(* Control logic *)
IF CtrlExton THEN
	REL_EN:=TRUE;
ELSE
	CASE CTRL_MODE OF
		 0: REL_EN:=FALSE;
		-1: REL_EN:=TRUE;
		-2: REL_EN:=CtrlKey;
		-3: REL_EN:=NOT CtrlKey;
		-4: REL_EN:=CtrlSens;
		-5: REL_EN:=NOT CtrlSens;
	ELSE
		IF CTRL_MODE>0 THEN
			REL_EN:=TrigTimer.Q;
			TrigTimer.PT:=T#1S*CTRL_MODE;
		ELSE
			REL_EN:=FALSE;
		END_IF
	END_CASE
END_IF

(* Temporary energy counter *)
TickTimer(IN:=NOT TickTimer.Q);
IF TickTimer.Q AND REL_EN THEN
	WORKINGTIME:=WORKINGTIME+1;
	ENERGYCOUNTER_T:=ENERGYCOUNTER_T+REL_V*REL_A;
	IF ENERGYCOUNTER_T>36000000 THEN
		ENERGYCOUNTER_T:=ENERGYCOUNTER_T-36000000;
		ENERGYCOUNTER:=ENERGYCOUNTER+1;		
	END_IF
END_IF

(* Generate status events *)
sREL_EN(IN:=REL_EN);
IF sREL_EN.EVL THEN LogEv(EL_Log,EO_LUXM,ID,2,''); END_IF
IF sREL_EN.EVH THEN LogEv(EL_Log,EO_LUXM,ID,3,''); POWERONCYCLES:=POWERONCYCLES+1; END_IF

(* Check status feedback *)
chkREL_ST(IN:=(REL_ST<>REL_EN));
IF chkREL_ST.EVH THEN LogEv(EL_Alarm,EO_LUXM,ID,9,''); END_IF
IF chkREL_ST.EVL AND sREL_ALM=0 THEN LogEv(EL_Log,EO_LUXM,ID,1,''); END_IF

(* Check controller alarm *)
IF sREL_ALM<>REL_ALM THEN
	CASE REL_ALM OF
		0: IF NOT chkREL_ST.OUT THEN LogEv(EL_Log,EO_LUXM,ID,1,''); END_IF
		1: LogEv(EL_Alarm,EO_LUXM,ID,6,'');
		2: LogEv(EL_Wrn  ,EO_LUXM,ID,4,WORD_TO_STRING(REL_A));
		3: LogEv(EL_Wrn  ,EO_LUXM,ID,5,WORD_TO_STRING(REL_A));
		4: LogEv(EL_Alarm,EO_LUXM,ID,7,WORD_TO_STRING(REL_A));
		5: LogEv(EL_Alarm,EO_LUXM,ID,8,'');
	END_CASE
	sREL_ALM:=REL_ALM;
END_IF

(* Status color *)
   IF REL_ALM=1 OR REL_ALM>3 OR chkREL_ST.OUT	THEN Status_Log:=2; Status_Vis:=COLOR_RED;
ELSIF REL_ALM<>0								THEN Status_Log:=1; Status_Vis:=COLOR_YELLOW;
                  	   							ELSE Status_Log:=0; Status_Vis:=SEL(REL_EN,COLOR_GREEN_OFF,COLOR_GREEN);
END_IF

ACTION AddLogData:
Logger.s1:=INSERT('&LUXM=',BYTE_TO_STRING(ID),5);
IF ID<10 THEN Logger.s1:=INSERT(Logger.s1,'0',5); END_IF

Logger.s1:=CONCAT(Logger.s1,WORD_TO_STRING(REL_V));				Logger.s1:=CONCAT(Logger.s1,';');
Logger.s1:=CONCAT(Logger.s1,WORD_TO_STRING(REL_A));				Logger.s1:=CONCAT(Logger.s1,';');
Logger.s1:=CONCAT(Logger.s1,DWORD_TO_STRING(ENERGYCOUNTER));	Logger.s1:=CONCAT(Logger.s1,';');
Logger.s1:=CONCAT(Logger.s1,DWORD_TO_STRING(WORKINGTIME));		Logger.s1:=CONCAT(Logger.s1,';');
Logger.s1:=CONCAT(Logger.s1,DWORD_TO_STRING(POWERONCYCLES));	Logger.s1:=CONCAT(Logger.s1,';');
Logger.s1:=CONCAT(Logger.s1,INT_TO_STRING(REL_TEMP));			Logger.s1:=CONCAT(Logger.s1,';');

Logger.s1:=CONCAT(Logger.s1,BYTE_TO_STRING(Status_Log));
ADDSTRING(ADR(Logger.TData), ADR(Logger.s1), Logger.TLen);
END_ACTION

ACTION StatReset:
(* Reset statistic counters *)
WORKINGTIME:=0;
POWERONCYCLES:=0;
ENERGYCOUNTER:=0;
END_ACTION

END_FUNCTION_BLOCK

// Utils Functions/DirOpen_FB
FUNCTION_BLOCK DirOpen_FB
VAR_INPUT
END_VAR
VAR_OUTPUT
END_VAR
VAR
	iFilesCount, counter : word;
//	DirNames: array[1..64] of string;
//	FileNames: array[1..64] of string;
	
	sDirName : STRING;
	sDirEntry : STRING;
	udiDirHandle : RTS_IEC_HANDLE;
	stDirInfo : DirInfo;
	udiResult : __XWORD;
	udiCreateError: UDINT;
	udiReadError: UDINT;
END_VAR

(*
sDirName:='Pippo';
udiCreateError := SysDirCreate(szDir:= sDirName);
*)

//ConfPath:='/media/sd/';	
sDirName:=CONCAT(STR1:=ConfPath, STR2:=sDirName);
udiDirHandle := SysDirOpen(szDir:= sDirName, szDirEntry:= sDirEntry, diMaxDirEntry:= 1024,
				pDirInfo:= ADR(stDirInfo), pResult:= udiResult);

(* Iterate through all direcotry entries and count them. The implicit entries with points are not count.
when the last entry is reached the SysDirRead always delivers the last entry.*)
iFilesCount := 0;
counter := 1;
repeat
	if FIND(sDirEntry, '.') <> 1 then
		iFilesCount := iFilesCount +1;
	end_if
	udiReadError:= SysDirRead(hDir:= udiDirHandle, szDirEntry:= sDirEntry, diMaxDirEntry:= 1024, pDirInfo:=ADR(stDirInfo) );
	// SysDirRead is used to Directory Info
	// Here, Im using SysDirRead to Find Folder Names within a Directory
	// If stDirInfo.diDirectory is Hex 2 , then the Directory is a folder, otherwise Hex 0 is a File
	if stDirInfo.diDirectory = 16#2 and Find(sDirEntry,'.') <> 1 then
		DirNames[counter]:=sDirEntry;
	else
		FileNames[counter]:=sDirEntry;
	counter:=counter+1;
	end_if
until 
	udiReadError = CmpErrors.Errors.ERR_END_OF_OBJECT
end_repeat

END_FUNCTION_BLOCK

// AC14nn/Application/VIS_CHONOEDITOR
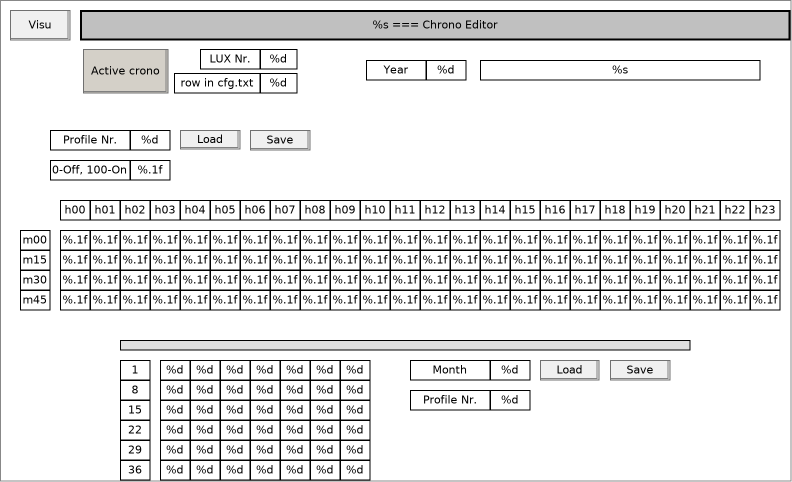
VISUALIZATION VIS_CHONOEDITOR  // 792x482
VAR_IN_OUT
//	x	: word;
//	LuxSel	: word;	
END_VAR
    Rectangle (200,49 60x20), "LUX Nr."
    Rectangle (260,49 37x20), "%d", text variable: CronEd.CN_Sel, colour toggle: CronEd.CN_Sel<>CronEd.CN_Act
        OnMouseDown: write the text variable via Edit, min 1, max 900, title '1'
    Rectangle (50,130 80x20), "Profile Nr."
    Rectangle (130,130 40x20), "%d", text variable: CronEd.PR_Sel, colour toggle: CronEd.PR_Sel<>CronEd.PR_Act
        OnMouseDown: write the text variable via Edit, min 1, max 10
    Rectangle (50,160 80x20), "0-Off, 100-On"
    Rectangle (130,160 40x20), "%.1f", text variable: CronEd.PR_TT
        OnMouseDown: write the text variable via Edit
    Button (180,130 60x19), "Load", pressed state: CronEd.PR_Load
        toggle CronEd.PR_Load
    Button (250,130 60x20), "Save", pressed state: CronEd.PR_Save
        toggle CronEd.PR_Save
    Rectangle (20,230 30x20), "m00"
    Rectangle (20,250 30x20), "m15"
    Rectangle (20,270 30x20), "m30"
    Rectangle (20,290 30x20), "m45"
    Rectangle (80,10 710x30), "%s === Chrono Editor", text variable: Plant_NAME
    Button (10,10 60x30), "Visu"
        OnMouseUp:  Assign=PLC_Visualization, Type=Assignment
    Polygon (20,210)
    RoundedRectangle (60,230 30x20), "%.1f", text variable: INT_TO_REAL(CronEd.PR.Setpoint[0])/10
        OnMouseUp: execute { CronEd.PR.Setpoint[0]:=(REAL_TO_WORD(CronEd.PR_TT*10)); }
    RoundedRectangle (60,250 30x20), "%.1f", text variable: INT_TO_REAL(CronEd.PR.Setpoint[1])/10
        OnMouseUp: execute { CronEd.PR.Setpoint[1]:=(REAL_TO_WORD(CronEd.PR_TT*10)); }
    RoundedRectangle (60,270 30x20), "%.1f", text variable: INT_TO_REAL(CronEd.PR.Setpoint[2])/10
        OnMouseUp: execute { CronEd.PR.Setpoint[2]:=(REAL_TO_WORD(CronEd.PR_TT*10)); }
    RoundedRectangle (60,290 30x20), "%.1f", text variable: INT_TO_REAL(CronEd.PR.Setpoint[3])/10
        OnMouseUp: execute { CronEd.PR.Setpoint[3]:=(REAL_TO_WORD(CronEd.PR_TT*10)); }
    Rectangle (60,200 30x20), "h00"
        OnMouseUp: execute { CronEd.PR.Setpoint[0]:=(REAL_TO_WORD(CronEd.PR_TT*10)); }
        OnMouseUp: execute { CronEd.PR.Setpoint[1]:=(REAL_TO_WORD(CronEd.PR_TT*10)); }
        OnMouseUp: execute { CronEd.PR.Setpoint[2]:=(REAL_TO_WORD(CronEd.PR_TT*10)); }
        OnMouseUp: execute { CronEd.PR.Setpoint[3]:=(REAL_TO_WORD(CronEd.PR_TT*10)); }
    RoundedRectangle (90,230 30x20), "%.1f", text variable: INT_TO_REAL(CronEd.PR.Setpoint[4])/10
        OnMouseUp: execute { CronEd.PR.Setpoint[4]:=(REAL_TO_WORD(CronEd.PR_TT*10)); }
    RoundedRectangle (90,250 30x20), "%.1f", text variable: INT_TO_REAL(CronEd.PR.Setpoint[5])/10
        OnMouseUp: execute { CronEd.PR.Setpoint[5]:=(REAL_TO_WORD(CronEd.PR_TT*10)); }
    RoundedRectangle (90,270 30x20), "%.1f", text variable: INT_TO_REAL(CronEd.PR.Setpoint[6])/10
        OnMouseUp: execute { CronEd.PR.Setpoint[6]:=(REAL_TO_WORD(CronEd.PR_TT*10)); }
    RoundedRectangle (90,290 30x20), "%.1f", text variable: INT_TO_REAL(CronEd.PR.Setpoint[7])/10
        OnMouseUp: execute { CronEd.PR.Setpoint[7]:=(REAL_TO_WORD(CronEd.PR_TT*10)); }
    Rectangle (90,200 30x20), "h01"
        OnMouseUp: execute { CronEd.PR.Setpoint[4]:=(REAL_TO_WORD(CronEd.PR_TT*10)); }
        OnMouseUp: execute { CronEd.PR.Setpoint[5]:=(REAL_TO_WORD(CronEd.PR_TT*10)); }
        OnMouseUp: execute { CronEd.PR.Setpoint[6]:=(REAL_TO_WORD(CronEd.PR_TT*10)); }
        OnMouseUp: execute { CronEd.PR.Setpoint[7]:=(REAL_TO_WORD(CronEd.PR_TT*10)); }
    RoundedRectangle (120,230 30x20), "%.1f", text variable: INT_TO_REAL(CronEd.PR.Setpoint[8])/10
        OnMouseUp: execute { CronEd.PR.Setpoint[8]:=(REAL_TO_WORD(CronEd.PR_TT*10)); }
    RoundedRectangle (120,250 30x20), "%.1f", text variable: INT_TO_REAL(CronEd.PR.Setpoint[9])/10
        OnMouseUp: execute { CronEd.PR.Setpoint[9]:=(REAL_TO_WORD(CronEd.PR_TT*10)); }
    RoundedRectangle (120,270 30x20), "%.1f", text variable: INT_TO_REAL(CronEd.PR.Setpoint[10])/10
        OnMouseUp: execute { CronEd.PR.Setpoint[10]:=(REAL_TO_WORD(CronEd.PR_TT*10)); }
    RoundedRectangle (120,290 30x20), "%.1f", text variable: INT_TO_REAL(CronEd.PR.Setpoint[11])/10
        OnMouseUp: execute { CronEd.PR.Setpoint[11]:=(REAL_TO_WORD(CronEd.PR_TT*10)); }
    Rectangle (120,200 30x20), "h02"
        OnMouseUp: execute { CronEd.PR.Setpoint[8]:=(REAL_TO_WORD(CronEd.PR_TT*10)); }
        OnMouseUp: execute { CronEd.PR.Setpoint[9]:=(REAL_TO_WORD(CronEd.PR_TT*10)); }
        OnMouseUp: execute { CronEd.PR.Setpoint[10]:=(REAL_TO_WORD(CronEd.PR_TT*10)); }
        OnMouseUp: execute { CronEd.PR.Setpoint[11]:=(REAL_TO_WORD(CronEd.PR_TT*10)); }
    RoundedRectangle (150,230 30x20), "%.1f", text variable: INT_TO_REAL(CronEd.PR.Setpoint[12])/10
        OnMouseUp: execute { CronEd.PR.Setpoint[12]:=(REAL_TO_WORD(CronEd.PR_TT*10)); }
    RoundedRectangle (150,250 30x20), "%.1f", text variable: INT_TO_REAL(CronEd.PR.Setpoint[13])/10
        OnMouseUp: execute { CronEd.PR.Setpoint[13]:=(REAL_TO_WORD(CronEd.PR_TT*10)); }
    RoundedRectangle (150,270 30x20), "%.1f", text variable: INT_TO_REAL(CronEd.PR.Setpoint[14])/10
        OnMouseUp: execute { CronEd.PR.Setpoint[14]:=(REAL_TO_WORD(CronEd.PR_TT*10)); }
    RoundedRectangle (150,290 30x20), "%.1f", text variable: INT_TO_REAL(CronEd.PR.Setpoint[15])/10
        OnMouseUp: execute { CronEd.PR.Setpoint[15]:=(REAL_TO_WORD(CronEd.PR_TT*10)); }
    Rectangle (150,200 30x20), "h03"
        OnMouseUp: execute { CronEd.PR.Setpoint[15]:=(REAL_TO_WORD(CronEd.PR_TT*10)); }
        OnMouseUp: execute { CronEd.PR.Setpoint[14]:=(REAL_TO_WORD(CronEd.PR_TT*10)); }
        OnMouseUp: execute { CronEd.PR.Setpoint[13]:=(REAL_TO_WORD(CronEd.PR_TT*10)); }
        OnMouseUp: execute { CronEd.PR.Setpoint[12]:=(REAL_TO_WORD(CronEd.PR_TT*10)); }
    RoundedRectangle (180,230 30x20), "%.1f", text variable: INT_TO_REAL(CronEd.PR.Setpoint[16])/10
        OnMouseUp: execute { CronEd.PR.Setpoint[16]:=(REAL_TO_WORD(CronEd.PR_TT*10)); }
    RoundedRectangle (180,250 30x20), "%.1f", text variable: INT_TO_REAL(CronEd.PR.Setpoint[17])/10
        OnMouseUp: execute { CronEd.PR.Setpoint[17]:=(REAL_TO_WORD(CronEd.PR_TT*10)); }
    RoundedRectangle (180,270 30x20), "%.1f", text variable: INT_TO_REAL(CronEd.PR.Setpoint[18])/10
        OnMouseUp: execute { CronEd.PR.Setpoint[18]:=(REAL_TO_WORD(CronEd.PR_TT*10)); }
    RoundedRectangle (180,290 30x20), "%.1f", text variable: INT_TO_REAL(CronEd.PR.Setpoint[19])/10
        OnMouseUp: execute { CronEd.PR.Setpoint[19]:=(REAL_TO_WORD(CronEd.PR_TT*10)); }
    Rectangle (180,200 30x20), "h04"
        OnMouseUp: execute { CronEd.PR.Setpoint[19]:=(REAL_TO_WORD(CronEd.PR_TT*10)); }
        OnMouseUp: execute { CronEd.PR.Setpoint[18]:=(REAL_TO_WORD(CronEd.PR_TT*10)); }
        OnMouseUp: execute { CronEd.PR.Setpoint[17]:=(REAL_TO_WORD(CronEd.PR_TT*10)); }
        OnMouseUp: execute { CronEd.PR.Setpoint[16]:=(REAL_TO_WORD(CronEd.PR_TT*10)); }
    RoundedRectangle (210,230 30x20), "%.1f", text variable: INT_TO_REAL(CronEd.PR.Setpoint[20])/10
        OnMouseUp: execute { CronEd.PR.Setpoint[20]:=(REAL_TO_WORD(CronEd.PR_TT*10)); }
    RoundedRectangle (210,250 30x20), "%.1f", text variable: INT_TO_REAL(CronEd.PR.Setpoint[21])/10
        OnMouseUp: execute { CronEd.PR.Setpoint[21]:=(REAL_TO_WORD(CronEd.PR_TT*10)); }
    RoundedRectangle (210,270 30x20), "%.1f", text variable: INT_TO_REAL(CronEd.PR.Setpoint[22])/10
        OnMouseUp: execute { CronEd.PR.Setpoint[22]:=(REAL_TO_WORD(CronEd.PR_TT*10)); }
    RoundedRectangle (210,290 30x20), "%.1f", text variable: INT_TO_REAL(CronEd.PR.Setpoint[23])/10
        OnMouseUp: execute { CronEd.PR.Setpoint[23]:=(REAL_TO_WORD(CronEd.PR_TT*10)); }
    Rectangle (210,200 30x20), "h05"
        OnMouseUp: execute { CronEd.PR.Setpoint[23]:=(REAL_TO_WORD(CronEd.PR_TT*10)); }
        OnMouseUp: execute { CronEd.PR.Setpoint[22]:=(REAL_TO_WORD(CronEd.PR_TT*10)); }
        OnMouseUp: execute { CronEd.PR.Setpoint[21]:=(REAL_TO_WORD(CronEd.PR_TT*10)); }
        OnMouseUp: execute { CronEd.PR.Setpoint[20]:=(REAL_TO_WORD(CronEd.PR_TT*10)); }
    RoundedRectangle (240,230 30x20), "%.1f", text variable: INT_TO_REAL(CronEd.PR.Setpoint[24])/10
        OnMouseUp: execute { CronEd.PR.Setpoint[24]:=(REAL_TO_WORD(CronEd.PR_TT*10)); }
    RoundedRectangle (240,250 30x20), "%.1f", text variable: INT_TO_REAL(CronEd.PR.Setpoint[25])/10
        OnMouseUp: execute { CronEd.PR.Setpoint[25]:=(REAL_TO_WORD(CronEd.PR_TT*10)); }
    RoundedRectangle (240,270 30x20), "%.1f", text variable: INT_TO_REAL(CronEd.PR.Setpoint[26])/10
        OnMouseUp: execute { CronEd.PR.Setpoint[26]:=(REAL_TO_WORD(CronEd.PR_TT*10)); }
    RoundedRectangle (240,290 30x20), "%.1f", text variable: INT_TO_REAL(CronEd.PR.Setpoint[27])/10
        OnMouseUp: execute { CronEd.PR.Setpoint[27]:=(REAL_TO_WORD(CronEd.PR_TT*10)); }
    Rectangle (240,200 30x20), "h06"
        OnMouseUp: execute { CronEd.PR.Setpoint[27]:=(REAL_TO_WORD(CronEd.PR_TT*10)); }
        OnMouseUp: execute { CronEd.PR.Setpoint[26]:=(REAL_TO_WORD(CronEd.PR_TT*10)); }
        OnMouseUp: execute { CronEd.PR.Setpoint[25]:=(REAL_TO_WORD(CronEd.PR_TT*10)); }
        OnMouseUp: execute { CronEd.PR.Setpoint[24]:=(REAL_TO_WORD(CronEd.PR_TT*10)); }
    RoundedRectangle (270,230 30x20), "%.1f", text variable: INT_TO_REAL(CronEd.PR.Setpoint[28])/10
        OnMouseUp: execute { CronEd.PR.Setpoint[28]:=(REAL_TO_WORD(CronEd.PR_TT*10)); }
    RoundedRectangle (270,250 30x20), "%.1f", text variable: INT_TO_REAL(CronEd.PR.Setpoint[29])/10
        OnMouseUp: execute { CronEd.PR.Setpoint[29]:=(REAL_TO_WORD(CronEd.PR_TT*10)); }
    RoundedRectangle (270,270 30x20), "%.1f", text variable: INT_TO_REAL(CronEd.PR.Setpoint[30])/10
        OnMouseUp: execute { CronEd.PR.Setpoint[30]:=(REAL_TO_WORD(CronEd.PR_TT*10)); }
    RoundedRectangle (270,290 30x20), "%.1f", text variable: INT_TO_REAL(CronEd.PR.Setpoint[31])/10
        OnMouseUp: execute { CronEd.PR.Setpoint[31]:=(REAL_TO_WORD(CronEd.PR_TT*10)); }
    Rectangle (270,200 30x20), "h07"
        OnMouseUp: execute { CronEd.PR.Setpoint[31]:=(REAL_TO_WORD(CronEd.PR_TT*10)); }
        OnMouseUp: execute { CronEd.PR.Setpoint[30]:=(REAL_TO_WORD(CronEd.PR_TT*10)); }
        OnMouseUp: execute { CronEd.PR.Setpoint[29]:=(REAL_TO_WORD(CronEd.PR_TT*10)); }
        OnMouseUp: execute { CronEd.PR.Setpoint[28]:=(REAL_TO_WORD(CronEd.PR_TT*10)); }
    RoundedRectangle (300,230 30x20), "%.1f", text variable: INT_TO_REAL(CronEd.PR.Setpoint[32])/10
        OnMouseUp: execute { CronEd.PR.Setpoint[32]:=(REAL_TO_WORD(CronEd.PR_TT*10)); }
    RoundedRectangle (300,250 30x20), "%.1f", text variable: INT_TO_REAL(CronEd.PR.Setpoint[33])/10
        OnMouseUp: execute { CronEd.PR.Setpoint[33]:=(REAL_TO_WORD(CronEd.PR_TT*10)); }
    RoundedRectangle (300,270 30x20), "%.1f", text variable: INT_TO_REAL(CronEd.PR.Setpoint[34])/10
        OnMouseUp: execute { CronEd.PR.Setpoint[34]:=(REAL_TO_WORD(CronEd.PR_TT*10)); }
    RoundedRectangle (300,290 30x20), "%.1f", text variable: INT_TO_REAL(CronEd.PR.Setpoint[35])/10
        OnMouseUp: execute { CronEd.PR.Setpoint[35]:=(REAL_TO_WORD(CronEd.PR_TT*10)); }
    Rectangle (300,200 30x20), "h08"
        OnMouseUp: execute { CronEd.PR.Setpoint[35]:=(REAL_TO_WORD(CronEd.PR_TT*10)); }
        OnMouseUp: execute { CronEd.PR.Setpoint[34]:=(REAL_TO_WORD(CronEd.PR_TT*10)); }
        OnMouseUp: execute { CronEd.PR.Setpoint[33]:=(REAL_TO_WORD(CronEd.PR_TT*10)); }
        OnMouseUp: execute { CronEd.PR.Setpoint[32]:=(REAL_TO_WORD(CronEd.PR_TT*10)); }
    RoundedRectangle (330,230 30x20), "%.1f", text variable: INT_TO_REAL(CronEd.PR.Setpoint[36])/10
        OnMouseUp: execute { CronEd.PR.Setpoint[36]:=(REAL_TO_WORD(CronEd.PR_TT*10)); }
    RoundedRectangle (330,250 30x20), "%.1f", text variable: INT_TO_REAL(CronEd.PR.Setpoint[37])/10
        OnMouseUp: execute { CronEd.PR.Setpoint[37]:=(REAL_TO_WORD(CronEd.PR_TT*10)); }
    RoundedRectangle (330,270 30x20), "%.1f", text variable: INT_TO_REAL(CronEd.PR.Setpoint[38])/10
        OnMouseUp: execute { CronEd.PR.Setpoint[38]:=(REAL_TO_WORD(CronEd.PR_TT*10)); }
    RoundedRectangle (330,290 30x20), "%.1f", text variable: INT_TO_REAL(CronEd.PR.Setpoint[39])/10
        OnMouseUp: execute { CronEd.PR.Setpoint[39]:=(REAL_TO_WORD(CronEd.PR_TT*10)); }
    Rectangle (330,200 30x20), "h09"
        OnMouseUp: execute { CronEd.PR.Setpoint[39]:=(REAL_TO_WORD(CronEd.PR_TT*10)); }
        OnMouseUp: execute { CronEd.PR.Setpoint[38]:=(REAL_TO_WORD(CronEd.PR_TT*10)); }
        OnMouseUp: execute { CronEd.PR.Setpoint[37]:=(REAL_TO_WORD(CronEd.PR_TT*10)); }
        OnMouseUp: execute { CronEd.PR.Setpoint[36]:=(REAL_TO_WORD(CronEd.PR_TT*10)); }
    RoundedRectangle (360,230 30x20), "%.1f", text variable: INT_TO_REAL(CronEd.PR.Setpoint[40])/10
        OnMouseUp: execute { CronEd.PR.Setpoint[40]:=(REAL_TO_WORD(CronEd.PR_TT*10)); }
    RoundedRectangle (360,250 30x20), "%.1f", text variable: INT_TO_REAL(CronEd.PR.Setpoint[41])/10
        OnMouseUp: execute { CronEd.PR.Setpoint[41]:=(REAL_TO_WORD(CronEd.PR_TT*10)); }
    RoundedRectangle (360,270 30x20), "%.1f", text variable: INT_TO_REAL(CronEd.PR.Setpoint[42])/10
        OnMouseUp: execute { CronEd.PR.Setpoint[42]:=(REAL_TO_WORD(CronEd.PR_TT*10)); }
    RoundedRectangle (360,290 30x20), "%.1f", text variable: INT_TO_REAL(CronEd.PR.Setpoint[43])/10
        OnMouseUp: execute { CronEd.PR.Setpoint[43]:=(REAL_TO_WORD(CronEd.PR_TT*10)); }
    Rectangle (360,200 30x20), "h10"
        OnMouseUp: execute { CronEd.PR.Setpoint[43]:=(REAL_TO_WORD(CronEd.PR_TT*10)); }
        OnMouseUp: execute { CronEd.PR.Setpoint[42]:=(REAL_TO_WORD(CronEd.PR_TT*10)); }
        OnMouseUp: execute { CronEd.PR.Setpoint[41]:=(REAL_TO_WORD(CronEd.PR_TT*10)); }
        OnMouseUp: execute { CronEd.PR.Setpoint[40]:=(REAL_TO_WORD(CronEd.PR_TT*10)); }
    RoundedRectangle (390,230 30x20), "%.1f", text variable: INT_TO_REAL(CronEd.PR.Setpoint[44])/10
        OnMouseUp: execute { CronEd.PR.Setpoint[44]:=(REAL_TO_WORD(CronEd.PR_TT*10)); }
    RoundedRectangle (390,250 30x20), "%.1f", text variable: INT_TO_REAL(CronEd.PR.Setpoint[45])/10
        OnMouseUp: execute { CronEd.PR.Setpoint[45]:=(REAL_TO_WORD(CronEd.PR_TT*10)); }
    RoundedRectangle (390,270 30x20), "%.1f", text variable: INT_TO_REAL(CronEd.PR.Setpoint[46])/10
        OnMouseUp: execute { CronEd.PR.Setpoint[46]:=(REAL_TO_WORD(CronEd.PR_TT*10)); }
    RoundedRectangle (390,290 30x20), "%.1f", text variable: INT_TO_REAL(CronEd.PR.Setpoint[47])/10
        OnMouseUp: execute { CronEd.PR.Setpoint[47]:=(REAL_TO_WORD(CronEd.PR_TT*10)); }
    Rectangle (390,200 30x20), "h11"
        OnMouseUp: execute { CronEd.PR.Setpoint[47]:=(REAL_TO_WORD(CronEd.PR_TT*10)); }
        OnMouseUp: execute { CronEd.PR.Setpoint[46]:=(REAL_TO_WORD(CronEd.PR_TT*10)); }
        OnMouseUp: execute { CronEd.PR.Setpoint[45]:=(REAL_TO_WORD(CronEd.PR_TT*10)); }
        OnMouseUp: execute { CronEd.PR.Setpoint[44]:=(REAL_TO_WORD(CronEd.PR_TT*10)); }
    RoundedRectangle (420,230 30x20), "%.1f", text variable: INT_TO_REAL(CronEd.PR.Setpoint[48])/10
        OnMouseUp: execute { CronEd.PR.Setpoint[48]:=(REAL_TO_WORD(CronEd.PR_TT*10)); }
    RoundedRectangle (420,250 30x20), "%.1f", text variable: INT_TO_REAL(CronEd.PR.Setpoint[49])/10
        OnMouseUp: execute { CronEd.PR.Setpoint[49]:=(REAL_TO_WORD(CronEd.PR_TT*10)); }
    RoundedRectangle (420,270 30x20), "%.1f", text variable: INT_TO_REAL(CronEd.PR.Setpoint[50])/10
        OnMouseUp: execute { CronEd.PR.Setpoint[50]:=(REAL_TO_WORD(CronEd.PR_TT*10)); }
    RoundedRectangle (420,290 30x20), "%.1f", text variable: INT_TO_REAL(CronEd.PR.Setpoint[51])/10
        OnMouseUp: execute { CronEd.PR.Setpoint[51]:=(REAL_TO_WORD(CronEd.PR_TT*10)); }
    Rectangle (420,200 30x20), "h12"
        OnMouseUp: execute { CronEd.PR.Setpoint[51]:=(REAL_TO_WORD(CronEd.PR_TT*10)); }
        OnMouseUp: execute { CronEd.PR.Setpoint[50]:=(REAL_TO_WORD(CronEd.PR_TT*10)); }
        OnMouseUp: execute { CronEd.PR.Setpoint[49]:=(REAL_TO_WORD(CronEd.PR_TT*10)); }
        OnMouseUp: execute { CronEd.PR.Setpoint[48]:=(REAL_TO_WORD(CronEd.PR_TT*10)); }
    RoundedRectangle (450,230 30x20), "%.1f", text variable: INT_TO_REAL(CronEd.PR.Setpoint[52])/10
        OnMouseUp: execute { CronEd.PR.Setpoint[52]:=(REAL_TO_WORD(CronEd.PR_TT*10)); }
    RoundedRectangle (450,250 30x20), "%.1f", text variable: INT_TO_REAL(CronEd.PR.Setpoint[53])/10
        OnMouseUp: execute { CronEd.PR.Setpoint[53]:=(REAL_TO_WORD(CronEd.PR_TT*10)); }
    RoundedRectangle (450,270 30x20), "%.1f", text variable: INT_TO_REAL(CronEd.PR.Setpoint[54])/10
        OnMouseUp: execute { CronEd.PR.Setpoint[54]:=(REAL_TO_WORD(CronEd.PR_TT*10)); }
    RoundedRectangle (450,290 30x20), "%.1f", text variable: INT_TO_REAL(CronEd.PR.Setpoint[55])/10
        OnMouseUp: execute { CronEd.PR.Setpoint[55]:=(REAL_TO_WORD(CronEd.PR_TT*10)); }
    Rectangle (450,200 30x20), "h13"
        OnMouseUp: execute { CronEd.PR.Setpoint[55]:=(REAL_TO_WORD(CronEd.PR_TT*10)); }
        OnMouseUp: execute { CronEd.PR.Setpoint[54]:=(REAL_TO_WORD(CronEd.PR_TT*10)); }
        OnMouseUp: execute { CronEd.PR.Setpoint[53]:=(REAL_TO_WORD(CronEd.PR_TT*10)); }
        OnMouseUp: execute { CronEd.PR.Setpoint[52]:=(REAL_TO_WORD(CronEd.PR_TT*10)); }
    RoundedRectangle (480,230 30x20), "%.1f", text variable: INT_TO_REAL(CronEd.PR.Setpoint[56])/10
        OnMouseUp: execute { CronEd.PR.Setpoint[56]:=(REAL_TO_WORD(CronEd.PR_TT*10)); }
    RoundedRectangle (480,250 30x20), "%.1f", text variable: INT_TO_REAL(CronEd.PR.Setpoint[57])/10
        OnMouseUp: execute { CronEd.PR.Setpoint[57]:=(REAL_TO_WORD(CronEd.PR_TT*10)); }
    RoundedRectangle (480,270 30x20), "%.1f", text variable: INT_TO_REAL(CronEd.PR.Setpoint[58])/10
        OnMouseUp: execute { CronEd.PR.Setpoint[58]:=(REAL_TO_WORD(CronEd.PR_TT*10)); }
    RoundedRectangle (480,290 30x20), "%.1f", text variable: INT_TO_REAL(CronEd.PR.Setpoint[59])/10
        OnMouseUp: execute { CronEd.PR.Setpoint[59]:=(REAL_TO_WORD(CronEd.PR_TT*10)); }
    Rectangle (480,200 30x20), "h14"
        OnMouseUp: execute { CronEd.PR.Setpoint[59]:=(REAL_TO_WORD(CronEd.PR_TT*10)); }
        OnMouseUp: execute { CronEd.PR.Setpoint[58]:=(REAL_TO_WORD(CronEd.PR_TT*10)); }
        OnMouseUp: execute { CronEd.PR.Setpoint[57]:=(REAL_TO_WORD(CronEd.PR_TT*10)); }
        OnMouseUp: execute { CronEd.PR.Setpoint[56]:=(REAL_TO_WORD(CronEd.PR_TT*10)); }
    RoundedRectangle (510,230 30x20), "%.1f", text variable: INT_TO_REAL(CronEd.PR.Setpoint[60])/10
        OnMouseUp: execute { CronEd.PR.Setpoint[60]:=(REAL_TO_WORD(CronEd.PR_TT*10)); }
    RoundedRectangle (510,250 30x20), "%.1f", text variable: INT_TO_REAL(CronEd.PR.Setpoint[61])/10
        OnMouseUp: execute { CronEd.PR.Setpoint[61]:=(REAL_TO_WORD(CronEd.PR_TT*10)); }
    RoundedRectangle (510,270 30x20), "%.1f", text variable: INT_TO_REAL(CronEd.PR.Setpoint[62])/10
        OnMouseUp: execute { CronEd.PR.Setpoint[62]:=(REAL_TO_WORD(CronEd.PR_TT*10)); }
    RoundedRectangle (510,290 30x20), "%.1f", text variable: INT_TO_REAL(CronEd.PR.Setpoint[63])/10
        OnMouseUp: execute { CronEd.PR.Setpoint[63]:=(REAL_TO_WORD(CronEd.PR_TT*10)); }
    Rectangle (510,200 30x20), "h15"
        OnMouseUp: execute { CronEd.PR.Setpoint[63]:=(REAL_TO_WORD(CronEd.PR_TT*10)); }
        OnMouseUp: execute { CronEd.PR.Setpoint[62]:=(REAL_TO_WORD(CronEd.PR_TT*10)); }
        OnMouseUp: execute { CronEd.PR.Setpoint[61]:=(REAL_TO_WORD(CronEd.PR_TT*10)); }
        OnMouseUp: execute { CronEd.PR.Setpoint[60]:=(REAL_TO_WORD(CronEd.PR_TT*10)); }
    RoundedRectangle (540,230 30x20), "%.1f", text variable: INT_TO_REAL(CronEd.PR.Setpoint[64])/10
        OnMouseUp: execute { CronEd.PR.Setpoint[64]:=(REAL_TO_WORD(CronEd.PR_TT*10)); }
    RoundedRectangle (540,250 30x20), "%.1f", text variable: INT_TO_REAL(CronEd.PR.Setpoint[65])/10
        OnMouseUp: execute { CronEd.PR.Setpoint[65]:=(REAL_TO_WORD(CronEd.PR_TT*10)); }
    RoundedRectangle (540,270 30x20), "%.1f", text variable: INT_TO_REAL(CronEd.PR.Setpoint[66])/10
        OnMouseUp: execute { CronEd.PR.Setpoint[66]:=(REAL_TO_WORD(CronEd.PR_TT*10)); }
    RoundedRectangle (540,290 30x20), "%.1f", text variable: INT_TO_REAL(CronEd.PR.Setpoint[67])/10
        OnMouseUp: execute { CronEd.PR.Setpoint[67]:=(REAL_TO_WORD(CronEd.PR_TT*10)); }
    Rectangle (540,200 30x20), "h16"
        OnMouseUp: execute { CronEd.PR.Setpoint[67]:=(REAL_TO_WORD(CronEd.PR_TT*10)); }
        OnMouseUp: execute { CronEd.PR.Setpoint[66]:=(REAL_TO_WORD(CronEd.PR_TT*10)); }
        OnMouseUp: execute { CronEd.PR.Setpoint[65]:=(REAL_TO_WORD(CronEd.PR_TT*10)); }
        OnMouseUp: execute { CronEd.PR.Setpoint[64]:=(REAL_TO_WORD(CronEd.PR_TT*10)); }
    RoundedRectangle (570,230 30x20), "%.1f", text variable: INT_TO_REAL(CronEd.PR.Setpoint[68])/10
        OnMouseUp: execute { CronEd.PR.Setpoint[68]:=(REAL_TO_WORD(CronEd.PR_TT*10)); }
    RoundedRectangle (570,250 30x20), "%.1f", text variable: INT_TO_REAL(CronEd.PR.Setpoint[69])/10
        OnMouseUp: execute { CronEd.PR.Setpoint[69]:=(REAL_TO_WORD(CronEd.PR_TT*10)); }
    RoundedRectangle (570,270 30x20), "%.1f", text variable: INT_TO_REAL(CronEd.PR.Setpoint[70])/10
        OnMouseUp: execute { CronEd.PR.Setpoint[70]:=(REAL_TO_WORD(CronEd.PR_TT*10)); }
    RoundedRectangle (570,290 30x20), "%.1f", text variable: INT_TO_REAL(CronEd.PR.Setpoint[71])/10
        OnMouseUp: execute { CronEd.PR.Setpoint[71]:=(REAL_TO_WORD(CronEd.PR_TT*10)); }
    Rectangle (570,200 30x20), "h17"
        OnMouseUp: execute { CronEd.PR.Setpoint[71]:=(REAL_TO_WORD(CronEd.PR_TT*10)); }
        OnMouseUp: execute { CronEd.PR.Setpoint[70]:=(REAL_TO_WORD(CronEd.PR_TT*10)); }
        OnMouseUp: execute { CronEd.PR.Setpoint[69]:=(REAL_TO_WORD(CronEd.PR_TT*10)); }
        OnMouseUp: execute { CronEd.PR.Setpoint[68]:=(REAL_TO_WORD(CronEd.PR_TT*10)); }
    RoundedRectangle (600,230 30x20), "%.1f", text variable: INT_TO_REAL(CronEd.PR.Setpoint[72])/10
        OnMouseUp: execute { CronEd.PR.Setpoint[72]:=(REAL_TO_WORD(CronEd.PR_TT*10)); }
    RoundedRectangle (600,250 30x20), "%.1f", text variable: INT_TO_REAL(CronEd.PR.Setpoint[73])/10
        OnMouseUp: execute { CronEd.PR.Setpoint[73]:=(REAL_TO_WORD(CronEd.PR_TT*10)); }
    RoundedRectangle (600,270 30x20), "%.1f", text variable: INT_TO_REAL(CronEd.PR.Setpoint[74])/10
        OnMouseUp: execute { CronEd.PR.Setpoint[74]:=(REAL_TO_WORD(CronEd.PR_TT*10)); }
    RoundedRectangle (600,290 30x20), "%.1f", text variable: INT_TO_REAL(CronEd.PR.Setpoint[75])/10
        OnMouseUp: execute { CronEd.PR.Setpoint[75]:=(REAL_TO_WORD(CronEd.PR_TT*10)); }
    Rectangle (600,200 30x20), "h18"
        OnMouseUp: execute { CronEd.PR.Setpoint[75]:=(REAL_TO_WORD(CronEd.PR_TT*10)); }
        OnMouseUp: execute { CronEd.PR.Setpoint[74]:=(REAL_TO_WORD(CronEd.PR_TT*10)); }
        OnMouseUp: execute { CronEd.PR.Setpoint[73]:=(REAL_TO_WORD(CronEd.PR_TT*10)); }
        OnMouseUp: execute { CronEd.PR.Setpoint[72]:=(REAL_TO_WORD(CronEd.PR_TT*10)); }
    RoundedRectangle (630,230 30x20), "%.1f", text variable: INT_TO_REAL(CronEd.PR.Setpoint[76])/10
        OnMouseUp: execute { CronEd.PR.Setpoint[76]:=(REAL_TO_WORD(CronEd.PR_TT*10)); }
    RoundedRectangle (630,250 30x20), "%.1f", text variable: INT_TO_REAL(CronEd.PR.Setpoint[77])/10
        OnMouseUp: execute { CronEd.PR.Setpoint[77]:=(REAL_TO_WORD(CronEd.PR_TT*10)); }
    RoundedRectangle (630,270 30x20), "%.1f", text variable: INT_TO_REAL(CronEd.PR.Setpoint[78])/10
        OnMouseUp: execute { CronEd.PR.Setpoint[78]:=(REAL_TO_WORD(CronEd.PR_TT*10)); }
    RoundedRectangle (630,290 30x20), "%.1f", text variable: INT_TO_REAL(CronEd.PR.Setpoint[79])/10
        OnMouseUp: execute { CronEd.PR.Setpoint[79]:=(REAL_TO_WORD(CronEd.PR_TT*10)); }
    Rectangle (630,200 30x20), "h19"
        OnMouseUp: execute { CronEd.PR.Setpoint[79]:=(REAL_TO_WORD(CronEd.PR_TT*10)); }
        OnMouseUp: execute { CronEd.PR.Setpoint[78]:=(REAL_TO_WORD(CronEd.PR_TT*10)); }
        OnMouseUp: execute { CronEd.PR.Setpoint[77]:=(REAL_TO_WORD(CronEd.PR_TT*10)); }
        OnMouseUp: execute { CronEd.PR.Setpoint[76]:=(REAL_TO_WORD(CronEd.PR_TT*10)); }
    RoundedRectangle (660,230 30x20), "%.1f", text variable: INT_TO_REAL(CronEd.PR.Setpoint[80])/10
        OnMouseUp: execute { CronEd.PR.Setpoint[80]:=(REAL_TO_WORD(CronEd.PR_TT*10)); }
    RoundedRectangle (660,250 30x20), "%.1f", text variable: INT_TO_REAL(CronEd.PR.Setpoint[81])/10
        OnMouseUp: execute { CronEd.PR.Setpoint[81]:=(REAL_TO_WORD(CronEd.PR_TT*10)); }
    RoundedRectangle (660,270 30x20), "%.1f", text variable: INT_TO_REAL(CronEd.PR.Setpoint[82])/10
        OnMouseUp: execute { CronEd.PR.Setpoint[82]:=(REAL_TO_WORD(CronEd.PR_TT*10)); }
    RoundedRectangle (660,290 30x20), "%.1f", text variable: INT_TO_REAL(CronEd.PR.Setpoint[83])/10
        OnMouseUp: execute { CronEd.PR.Setpoint[83]:=(REAL_TO_WORD(CronEd.PR_TT*10)); }
    Rectangle (660,200 30x20), "h20"
        OnMouseUp: execute { CronEd.PR.Setpoint[83]:=(REAL_TO_WORD(CronEd.PR_TT*10)); }
        OnMouseUp: execute { CronEd.PR.Setpoint[82]:=(REAL_TO_WORD(CronEd.PR_TT*10)); }
        OnMouseUp: execute { CronEd.PR.Setpoint[81]:=(REAL_TO_WORD(CronEd.PR_TT*10)); }
        OnMouseUp: execute { CronEd.PR.Setpoint[80]:=(REAL_TO_WORD(CronEd.PR_TT*10)); }
    RoundedRectangle (690,230 30x20), "%.1f", text variable: INT_TO_REAL(CronEd.PR.Setpoint[84])/10
        OnMouseUp: execute { CronEd.PR.Setpoint[84]:=(REAL_TO_WORD(CronEd.PR_TT*10)); }
    RoundedRectangle (690,250 30x20), "%.1f", text variable: INT_TO_REAL(CronEd.PR.Setpoint[85])/10
        OnMouseUp: execute { CronEd.PR.Setpoint[85]:=(REAL_TO_WORD(CronEd.PR_TT*10)); }
    RoundedRectangle (690,270 30x20), "%.1f", text variable: INT_TO_REAL(CronEd.PR.Setpoint[86])/10
        OnMouseUp: execute { CronEd.PR.Setpoint[86]:=(REAL_TO_WORD(CronEd.PR_TT*10)); }
    RoundedRectangle (690,290 30x20), "%.1f", text variable: INT_TO_REAL(CronEd.PR.Setpoint[87])/10
        OnMouseUp: execute { CronEd.PR.Setpoint[87]:=(REAL_TO_WORD(CronEd.PR_TT*10)); }
    Rectangle (690,200 30x20), "h21"
        OnMouseUp: execute { CronEd.PR.Setpoint[87]:=(REAL_TO_WORD(CronEd.PR_TT*10)); }
        OnMouseUp: execute { CronEd.PR.Setpoint[86]:=(REAL_TO_WORD(CronEd.PR_TT*10)); }
        OnMouseUp: execute { CronEd.PR.Setpoint[85]:=(REAL_TO_WORD(CronEd.PR_TT*10)); }
        OnMouseUp: execute { CronEd.PR.Setpoint[84]:=(REAL_TO_WORD(CronEd.PR_TT*10)); }
    RoundedRectangle (720,230 30x20), "%.1f", text variable: INT_TO_REAL(CronEd.PR.Setpoint[88])/10
        OnMouseUp: execute { CronEd.PR.Setpoint[88]:=(REAL_TO_WORD(CronEd.PR_TT*10)); }
    RoundedRectangle (720,250 30x20), "%.1f", text variable: INT_TO_REAL(CronEd.PR.Setpoint[89])/10
        OnMouseUp: execute { CronEd.PR.Setpoint[89]:=(REAL_TO_WORD(CronEd.PR_TT*10)); }
    RoundedRectangle (720,270 30x20), "%.1f", text variable: INT_TO_REAL(CronEd.PR.Setpoint[90])/10
        OnMouseUp: execute { CronEd.PR.Setpoint[90]:=(REAL_TO_WORD(CronEd.PR_TT*10)); }
    RoundedRectangle (720,290 30x20), "%.1f", text variable: INT_TO_REAL(CronEd.PR.Setpoint[91])/10
        OnMouseUp: execute { CronEd.PR.Setpoint[91]:=(REAL_TO_WORD(CronEd.PR_TT*10)); }
    Rectangle (720,200 30x20), "h22"
        OnMouseUp: execute { CronEd.PR.Setpoint[91]:=(REAL_TO_WORD(CronEd.PR_TT*10)); }
        OnMouseUp: execute { CronEd.PR.Setpoint[90]:=(REAL_TO_WORD(CronEd.PR_TT*10)); }
        OnMouseUp: execute { CronEd.PR.Setpoint[89]:=(REAL_TO_WORD(CronEd.PR_TT*10)); }
        OnMouseUp: execute { CronEd.PR.Setpoint[88]:=(REAL_TO_WORD(CronEd.PR_TT*10)); }
    RoundedRectangle (750,230 30x20), "%.1f", text variable: INT_TO_REAL(CronEd.PR.Setpoint[92])/10
        OnMouseUp: execute { CronEd.PR.Setpoint[92]:=(REAL_TO_WORD(CronEd.PR_TT*10)); }
    RoundedRectangle (750,250 30x20), "%.1f", text variable: INT_TO_REAL(CronEd.PR.Setpoint[93])/10
        OnMouseUp: execute { CronEd.PR.Setpoint[93]:=(REAL_TO_WORD(CronEd.PR_TT*10)); }
    RoundedRectangle (750,270 30x20), "%.1f", text variable: INT_TO_REAL(CronEd.PR.Setpoint[94])/10
        OnMouseUp: execute { CronEd.PR.Setpoint[94]:=(REAL_TO_WORD(CronEd.PR_TT*10)); }
    RoundedRectangle (750,290 30x20), "%.1f", text variable: INT_TO_REAL(CronEd.PR.Setpoint[95])/10
        OnMouseUp: execute { CronEd.PR.Setpoint[95]:=(REAL_TO_WORD(CronEd.PR_TT*10)); }
    Rectangle (750,200 30x20), "h23"
        OnMouseUp: execute { CronEd.PR.Setpoint[95]:=(REAL_TO_WORD(CronEd.PR_TT*10)); }
        OnMouseUp: execute { CronEd.PR.Setpoint[94]:=(REAL_TO_WORD(CronEd.PR_TT*10)); }
        OnMouseUp: execute { CronEd.PR.Setpoint[93]:=(REAL_TO_WORD(CronEd.PR_TT*10)); }
        OnMouseUp: execute { CronEd.PR.Setpoint[92]:=(REAL_TO_WORD(CronEd.PR_TT*10)); }
    Rectangle (410,360 80x20), "Month"
    Rectangle (490,360 40x20), "%d", text variable: CronEd.CA_Sel, colour toggle: CronEd.CA_Sel<>CronEd.CA_Act
        OnMouseDown: write the text variable via Edit, min 1, max 12
    Rectangle (410,390 80x20), "Profile Nr."
    Rectangle (490,390 40x20), "%d", text variable: CronEd.CA_TPR
        OnMouseDown: write the text variable via Edit, min 0, max 10
    Button (540,360 59x20), "Load", pressed state: CronEd.CA_Load
        toggle CronEd.CA_Load
    Button (610,360 60x20), "Save", pressed state: CronEd.CA_Save
        toggle CronEd.CA_Save
    RoundedRectangle (160,360 30x20), "%d", text variable: CronEd.CA.Profile[0], colour toggle: CronEd.CA.Profile[0]=0, invisible if: CronEd.CA_DayF>0
        OnMouseUp: execute { CronEd.CA.Profile[0]:=(CronEd.CA_TPR); }
    Rectangle (120,360 30x20), "1"
    RoundedRectangle (190,360 30x20), "%d", text variable: CronEd.CA.Profile[1], colour toggle: CronEd.CA.Profile[1]=0, invisible if: CronEd.CA_DayF>1
        OnMouseUp: execute { CronEd.CA.Profile[1]:=(CronEd.CA_TPR); }
    RoundedRectangle (220,360 30x20), "%d", text variable: CronEd.CA.Profile[2], colour toggle: CronEd.CA.Profile[2]=0, invisible if: CronEd.CA_DayF>2
        OnMouseUp: execute { CronEd.CA.Profile[2]:=(CronEd.CA_TPR); }
    RoundedRectangle (250,360 30x20), "%d", text variable: CronEd.CA.Profile[3], colour toggle: CronEd.CA.Profile[3]=0, invisible if: CronEd.CA_DayF>3
        OnMouseUp: execute { CronEd.CA.Profile[3]:=(CronEd.CA_TPR); }
    RoundedRectangle (280,360 30x20), "%d", text variable: CronEd.CA.Profile[4], colour toggle: CronEd.CA.Profile[4]=0, invisible if: CronEd.CA_DayF>4
        OnMouseUp: execute { CronEd.CA.Profile[4]:=(CronEd.CA_TPR); }
    RoundedRectangle (310,360 30x20), "%d", text variable: CronEd.CA.Profile[5], colour toggle: CronEd.CA.Profile[5]=0, invisible if: CronEd.CA_DayF>5
        OnMouseUp: execute { CronEd.CA.Profile[5]:=(CronEd.CA_TPR); }
    RoundedRectangle (340,360 30x20), "%d", text variable: CronEd.CA.Profile[6], colour toggle: CronEd.CA.Profile[6]=0
        OnMouseUp: execute { CronEd.CA.Profile[6]:=(CronEd.CA_TPR); }
    RoundedRectangle (160,380 30x20), "%d", text variable: CronEd.CA.Profile[7], colour toggle: CronEd.CA.Profile[7]=0
        OnMouseUp: execute { CronEd.CA.Profile[7]:=(CronEd.CA_TPR); }
    Rectangle (120,380 30x20), "8"
    RoundedRectangle (190,380 30x20), "%d", text variable: CronEd.CA.Profile[8], colour toggle: CronEd.CA.Profile[8]=0
        OnMouseUp: execute { CronEd.CA.Profile[8]:=(CronEd.CA_TPR); }
    RoundedRectangle (220,380 30x20), "%d", text variable: CronEd.CA.Profile[9], colour toggle: CronEd.CA.Profile[9]=0
        OnMouseUp: execute { CronEd.CA.Profile[9]:=(CronEd.CA_TPR); }
    RoundedRectangle (250,380 30x20), "%d", text variable: CronEd.CA.Profile[10], colour toggle: CronEd.CA.Profile[10]=0
        OnMouseUp: execute { CronEd.CA.Profile[10]:=(CronEd.CA_TPR); }
    RoundedRectangle (280,380 30x20), "%d", text variable: CronEd.CA.Profile[11], colour toggle: CronEd.CA.Profile[11]=0
        OnMouseUp: execute { CronEd.CA.Profile[11]:=(CronEd.CA_TPR); }
    RoundedRectangle (310,380 30x20), "%d", text variable: CronEd.CA.Profile[12], colour toggle: CronEd.CA.Profile[12]=0
        OnMouseUp: execute { CronEd.CA.Profile[12]:=(CronEd.CA_TPR); }
    RoundedRectangle (340,380 30x20), "%d", text variable: CronEd.CA.Profile[13], colour toggle: CronEd.CA.Profile[13]=0
        OnMouseUp: execute { CronEd.CA.Profile[13]:=(CronEd.CA_TPR); }
    RoundedRectangle (160,400 30x20), "%d", text variable: CronEd.CA.Profile[14], colour toggle: CronEd.CA.Profile[14]=0
        OnMouseUp: execute { CronEd.CA.Profile[14]:=(CronEd.CA_TPR); }
    Rectangle (120,400 30x20), "15"
    RoundedRectangle (190,400 30x20), "%d", text variable: CronEd.CA.Profile[15], colour toggle: CronEd.CA.Profile[15]=0
        OnMouseUp: execute { CronEd.CA.Profile[15]:=(CronEd.CA_TPR); }
    RoundedRectangle (220,400 30x20), "%d", text variable: CronEd.CA.Profile[16], colour toggle: CronEd.CA.Profile[16]=0
        OnMouseUp: execute { CronEd.CA.Profile[16]:=(CronEd.CA_TPR); }
    RoundedRectangle (250,400 30x20), "%d", text variable: CronEd.CA.Profile[17], colour toggle: CronEd.CA.Profile[17]=0
        OnMouseUp: execute { CronEd.CA.Profile[17]:=(CronEd.CA_TPR); }
    RoundedRectangle (280,400 30x20), "%d", text variable: CronEd.CA.Profile[18], colour toggle: CronEd.CA.Profile[18]=0
        OnMouseUp: execute { CronEd.CA.Profile[18]:=(CronEd.CA_TPR); }
    RoundedRectangle (310,400 30x20), "%d", text variable: CronEd.CA.Profile[19], colour toggle: CronEd.CA.Profile[19]=0
        OnMouseUp: execute { CronEd.CA.Profile[19]:=(CronEd.CA_TPR); }
    RoundedRectangle (340,400 30x20), "%d", text variable: CronEd.CA.Profile[20], colour toggle: CronEd.CA.Profile[20]=0
        OnMouseUp: execute { CronEd.CA.Profile[20]:=(CronEd.CA_TPR); }
    RoundedRectangle (160,420 30x20), "%d", text variable: CronEd.CA.Profile[21], colour toggle: CronEd.CA.Profile[21]=0
        OnMouseUp: execute { CronEd.CA.Profile[21]:=(CronEd.CA_TPR); }
    Rectangle (120,420 30x20), "22"
    RoundedRectangle (190,420 30x20), "%d", text variable: CronEd.CA.Profile[22], colour toggle: CronEd.CA.Profile[22]=0
        OnMouseUp: execute { CronEd.CA.Profile[22]:=(CronEd.CA_TPR); }
    RoundedRectangle (220,420 30x20), "%d", text variable: CronEd.CA.Profile[23], colour toggle: CronEd.CA.Profile[23]=0
        OnMouseUp: execute { CronEd.CA.Profile[23]:=(CronEd.CA_TPR); }
    RoundedRectangle (250,420 30x20), "%d", text variable: CronEd.CA.Profile[24], colour toggle: CronEd.CA.Profile[24]=0
        OnMouseUp: execute { CronEd.CA.Profile[24]:=(CronEd.CA_TPR); }
    RoundedRectangle (280,420 30x20), "%d", text variable: CronEd.CA.Profile[25], colour toggle: CronEd.CA.Profile[25]=0
        OnMouseUp: execute { CronEd.CA.Profile[25]:=(CronEd.CA_TPR); }
    RoundedRectangle (310,420 30x20), "%d", text variable: CronEd.CA.Profile[26], colour toggle: CronEd.CA.Profile[26]=0
        OnMouseUp: execute { CronEd.CA.Profile[26]:=(CronEd.CA_TPR); }
    RoundedRectangle (340,420 30x20), "%d", text variable: CronEd.CA.Profile[27], colour toggle: CronEd.CA.Profile[27]=0
        OnMouseUp: execute { CronEd.CA.Profile[27]:=(CronEd.CA_TPR); }
    RoundedRectangle (160,440 30x20), "%d", text variable: CronEd.CA.Profile[28], colour toggle: CronEd.CA.Profile[28]=0
        OnMouseUp: execute { CronEd.CA.Profile[28]:=(CronEd.CA_TPR); }
    Rectangle (120,440 30x20), "29"
    RoundedRectangle (190,440 30x20), "%d", text variable: CronEd.CA.Profile[29], colour toggle: CronEd.CA.Profile[29]=0
        OnMouseUp: execute { CronEd.CA.Profile[29]:=(CronEd.CA_TPR); }
    RoundedRectangle (220,440 30x20), "%d", text variable: CronEd.CA.Profile[30], colour toggle: CronEd.CA.Profile[30]=0
        OnMouseUp: execute { CronEd.CA.Profile[30]:=(CronEd.CA_TPR); }
    RoundedRectangle (250,440 30x20), "%d", text variable: CronEd.CA.Profile[31], colour toggle: CronEd.CA.Profile[31]=0
        OnMouseUp: execute { CronEd.CA.Profile[31]:=(CronEd.CA_TPR); }
    RoundedRectangle (280,440 30x20), "%d", text variable: CronEd.CA.Profile[32], colour toggle: CronEd.CA.Profile[32]=0, invisible if: CronEd.CA_DayL<32
        OnMouseUp: execute { CronEd.CA.Profile[32]:=(CronEd.CA_TPR); }
    RoundedRectangle (310,440 30x20), "%d", text variable: CronEd.CA.Profile[33], colour toggle: CronEd.CA.Profile[33]=0, invisible if: CronEd.CA_DayL<33
        OnMouseUp: execute { CronEd.CA.Profile[33]:=(CronEd.CA_TPR); }
    RoundedRectangle (340,440 30x20), "%d", text variable: CronEd.CA.Profile[34], colour toggle: CronEd.CA.Profile[34]=0, invisible if: CronEd.CA_DayL<34
        OnMouseUp: execute { CronEd.CA.Profile[34]:=(CronEd.CA_TPR); }
    RoundedRectangle (160,460 30x20), "%d", text variable: CronEd.CA.Profile[35], colour toggle: CronEd.CA.Profile[35]=0, invisible if: CronEd.CA_DayL<35
        OnMouseUp: execute { CronEd.CA.Profile[35]:=(CronEd.CA_TPR); }
    Rectangle (120,460 30x20), "36", invisible if: CronEd.CA_DayL<35
    RoundedRectangle (190,460 30x20), "%d", text variable: CronEd.CA.Profile[36], colour toggle: CronEd.CA.Profile[36]=0, invisible if: CronEd.CA_DayL<36
        OnMouseUp: execute { CronEd.CA.Profile[36]:=(CronEd.CA_TPR); }
    RoundedRectangle (220,460 30x20), "%d", text variable: CronEd.CA.Profile[37], colour toggle: CronEd.CA.Profile[37]=0, invisible if: CronEd.CA_DayL<37
        OnMouseUp: execute { CronEd.CA.Profile[37]:=(CronEd.CA_TPR); }
    RoundedRectangle (250,460 30x20), "%d", text variable: CronEd.CA.Profile[38], colour toggle: CronEd.CA.Profile[38]=0, invisible if: CronEd.CA_DayL<38
        OnMouseUp: execute { CronEd.CA.Profile[38]:=(CronEd.CA_TPR); }
    RoundedRectangle (280,460 30x20), "%d", text variable: CronEd.CA.Profile[39], colour toggle: CronEd.CA.Profile[39]=0, invisible if: CronEd.CA_DayL<39
        OnMouseUp: execute { CronEd.CA.Profile[39]:=(CronEd.CA_TPR); }
    RoundedRectangle (310,460 30x20), "%d", text variable: CronEd.CA.Profile[40], colour toggle: CronEd.CA.Profile[40]=0, invisible if: CronEd.CA_DayL<40
        OnMouseUp: execute { CronEd.CA.Profile[40]:=(CronEd.CA_TPR); }
    RoundedRectangle (340,460 30x20), "%d", text variable: CronEd.CA.Profile[41], colour toggle: CronEd.CA.Profile[41]=0, invisible if: CronEd.CA_DayL<41
        OnMouseUp: execute { CronEd.CA.Profile[41]:=(CronEd.CA_TPR); }
    Rectangle (366,60 60x20), "Year"
    Rectangle (426,60 40x20), "%d", text variable: CronEd.CN_YSel, colour toggle: CronEd.CN_YSel<>CronEd.CN_YAct
        OnMouseDown: write the text variable via Edit, min 2000, max 2100, title '1'
    Rectangle (120,340 570x10)
    Rectangle (480,60 280x20), "%s", text variable: CronEd.Message
    Button (83,49 85x44), "Active crono"
        OnMouseClick: execute {
            CRON[CronEd.CN_Act].InitOK:=FALSE;
            (*	for x:= 1 to CRON_MAX do
            		if LuxElement[x].ID = CronEd.CN_Sel then
            			CronEd.CN_Act:=x;
            			CRON[CronEd.CN_Act].InitOK:=FALSE;
            			x:= CRON_MAX;
            		end_if
            	end_for
            *)
        }
    Rectangle (260,73 37x20), "%d", text variable: CronEd.CN_Act, colour toggle: CronEd.CN_Sel<>CronEd.CN_Act, invisible if: CronEd.Invisible
    Rectangle (174,73 86x20), "row in cfg.txt"
END_VISUALIZATION

// AC14nn/Application/PLC_FileManager
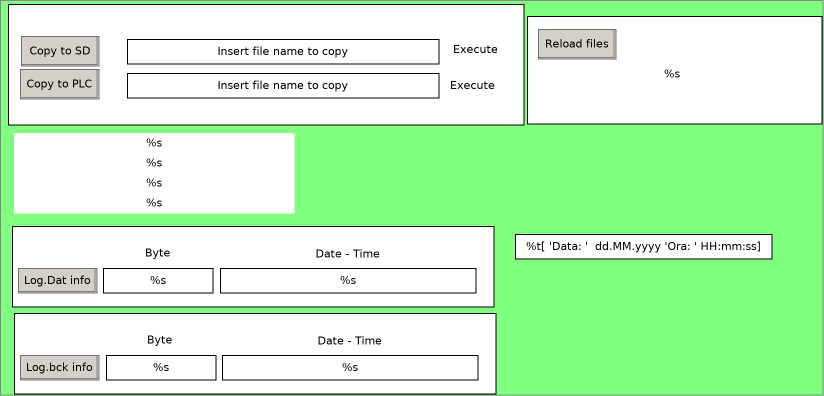
VISUALIZATION PLC_FileManager  // 824x396
    RoundedRectangle (12,226 482x81)
    RoundedRectangle (527,16 295x108)
    RoundedRectangle (8,4 516x121)
    Button (21,36 78x30), "Copy to SD"
        OnMouseClick:  ToggleVariable=PLC_PRG.CopyToSd
    Rectangle (127,39 312x25), "Insert file name to copy", text variable: PLC_PRG.FileCopyToSD.SourceFile
        OnMouseClick:  ToggleVariable=PLC_PRG.FileCopyToSD.FileCopying
        OnMouseUp: write the text variable via Edit
    Label (447,39 57x21), "Execute", invisible if: not(PLC_PRG.FileCopyToSD.FileCopying)
    Rectangle (127,73 312x25), "Insert file name to copy", text variable: PLC_PRG.FileCopySDToPLC.SourceFile
        OnMouseClick:  ToggleVariable=PLC_PRG.FileCopySDToPLC.FileCopying
        OnMouseUp: write the text variable via Edit
    Button (20,69 79x30), "Copy to PLC"
        OnMouseClick:  ToggleVariable=PLC_PRG.CopyToPLC
    Label (444,75 57x21), "Execute", invisible if: not(PLC_PRG.FileCopySDToPLC.FileCopying)
    Rectangle (14,133 280x20), "%s", text variable: PLC_PRG.OpenFileASI_PSG.Message
    Rectangle (14,153 280x20), "%s", text variable: PLC_PRG.OpenFileASI_LUX.Message
    Rectangle (14,173 280x20), "%s", text variable: PLC_PRG.OpenFileLUX_PSG.Message
    Rectangle (14,193 280x20), "%s", text variable: PLC_PRG.OpenFiles_Default_LUX.Message
    Button (538,29 78x30), "Reload files"
        OnMouseClick:  ToggleVariable=PLC_PRG.ReLoadFiles
    Rectangle (538,64 268x20), "%s", text variable: PLC_PRG.Message
    Button (18,268 79x25), "Log.Dat info"
        OnMouseClick:  ToggleVariable=PLC_PRG.FileTime
    Rectangle (220,268 256x25), "%s", text variable: PLC_PRG.FileSize_and_Time.LastModifyS
    Rectangle (103,268 110x25), "%s", text variable: PLC_PRG.FileSize_and_Time.Message
    Rectangle (103,243 110x20), "Byte"
    Rectangle (220,244 256x20), "Date - Time"
    Rectangle (515,234 257x25), "%t[ 'Data: ' dd.MM.yyyy 'Ora: ' HH:mm:ss]"
    RoundedRectangle (14,313 482x81)
    Button (20,355 79x25), "Log.bck info"
        OnMouseClick:  ToggleVariable=PLC_PRG.FileTime
    Rectangle (222,355 256x25), "%s", text variable: PLC_PRG.FileSize_and_Time.LastModifySBK
    Rectangle (105,330 110x20), "Byte"
    Rectangle (222,331 256x20), "Date - Time"
    Rectangle (106,355 110x25), "%s", text variable: PLC_PRG.FileSize_and_Time.MessageBK
END_VISUALIZATION

// AC14nn/Application/PLC_Visualization
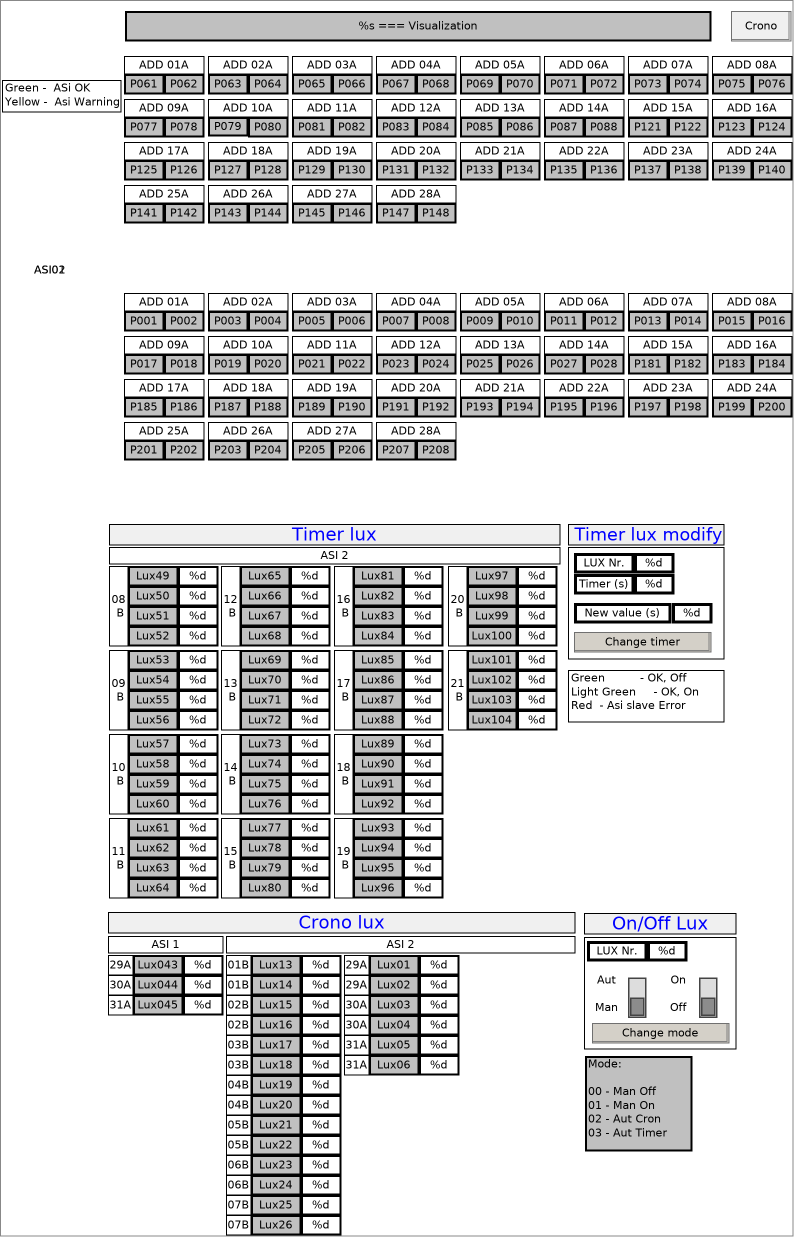
VISUALIZATION PLC_Visualization  // 794x1237
    Polygon (50,270), "ASI01", colour variable: ASI01.Status_Vis
    Polygon (50,270), "ASI02", colour variable: ASI02.Status_Vis
    Rectangle (124,293 80x18), "ADD 01A", colour toggle: ASI02.Asi_DeviceA[1]
    Rectangle (208,293 80x18), "ADD 02A", colour toggle: ASI02.Asi_DeviceA[2]
    Rectangle (292,293 80x18), "ADD 03A", colour toggle: ASI02.Asi_DeviceA[3]
    Rectangle (376,293 80x18), "ADD 04A", colour toggle: ASI02.Asi_DeviceA[4]
    Rectangle (460,293 80x18), "ADD 05A", colour toggle: ASI02.Asi_DeviceA[5]
    Rectangle (544,293 80x18), "ADD 06A", colour toggle: ASI02.Asi_DeviceA[6]
    Rectangle (628,293 80x18), "ADD 07A", colour toggle: ASI02.Asi_DeviceA[7]
    Rectangle (712,293 80x18), "ADD 08A", colour toggle: ASI02.Asi_DeviceA[8]
    Rectangle (124,336 80x18), "ADD 09A", colour toggle: ASI02.Asi_DeviceA[9]
    Rectangle (208,336 80x18), "ADD 10A", colour toggle: ASI02.Asi_DeviceA[10]
    Rectangle (292,336 80x18), "ADD 11A", colour toggle: ASI02.Asi_DeviceA[11]
    Rectangle (376,336 80x18), "ADD 12A", colour toggle: ASI02.Asi_DeviceA[12]
    Rectangle (460,336 80x18), "ADD 13A", colour toggle: ASI02.Asi_DeviceA[13]
    Rectangle (544,336 80x18), "ADD 14A", colour toggle: ASI02.Asi_DeviceA[14]
    Rectangle (628,336 80x18), "ADD 15A", colour toggle: ASI02.Asi_DeviceA[15]
    Rectangle (712,336 80x18), "ADD 16A", colour toggle: ASI02.Asi_DeviceA[16]
    Rectangle (124,379 80x18), "ADD 17A", colour toggle: ASI02.Asi_DeviceA[17]
    Rectangle (208,379 80x18), "ADD 18A", colour toggle: ASI02.Asi_DeviceA[18]
    Rectangle (292,379 80x18), "ADD 19A", colour toggle: ASI02.Asi_DeviceA[19]
    Rectangle (376,379 80x18), "ADD 20A", colour toggle: ASI02.Asi_DeviceA[20]
    Rectangle (460,379 80x18), "ADD 21A", colour toggle: ASI02.Asi_DeviceA[21]
    Rectangle (544,379 80x18), "ADD 22A", colour toggle: ASI02.Asi_DeviceA[22]
    Rectangle (628,379 80x18), "ADD 23A", colour toggle: ASI02.Asi_DeviceA[23]
    Rectangle (712,379 80x18), "ADD 24A", colour toggle: ASI02.Asi_DeviceA[24]
    Rectangle (124,422 80x18), "ADD 25A", colour toggle: ASI02.Asi_DeviceA[25]
    Rectangle (208,422 80x18), "ADD 26A", colour toggle: ASI02.Asi_DeviceA[26]
    Rectangle (292,422 80x18), "ADD 27A", colour toggle: ASI02.Asi_DeviceA[27]
    Rectangle (124,74 40x20), "P061", colour variable: DataPsgForVis[61].VisStatus
    Rectangle (164,74 40x20), "P062", colour variable: DataPsgForVis[62].VisStatus
    Rectangle (208,74 40x20), "P063", colour variable: DataPsgForVis[63].VisStatus
    Rectangle (248,74 40x20), "P064", colour variable: DataPsgForVis[64].VisStatus
    Rectangle (292,74 40x20), "P065", colour variable: DataPsgForVis[65].VisStatus
    Rectangle (332,74 40x20), "P066", colour variable: DataPsgForVis[66].VisStatus
    Rectangle (376,74 40x20), "P067", colour variable: DataPsgForVis[67].VisStatus
    Rectangle (416,74 40x20), "P068", colour variable: DataPsgForVis[68].VisStatus
    Rectangle (460,74 40x20), "P069", colour variable: DataPsgForVis[69].VisStatus
    Rectangle (500,74 40x20), "P070", colour variable: DataPsgForVis[70].VisStatus
    Rectangle (544,74 40x20), "P071", colour variable: DataPsgForVis[71].VisStatus
    Rectangle (584,74 40x20), "P072", colour variable: DataPsgForVis[72].VisStatus
    Rectangle (628,74 40x20), "P073", colour variable: DataPsgForVis[73].VisStatus
    Rectangle (668,74 40x20), "P074", colour variable: DataPsgForVis[74].VisStatus
    Rectangle (712,74 40x20), "P075", colour variable: DataPsgForVis[75].VisStatus
    Rectangle (752,74 40x20), "P076", colour variable: DataPsgForVis[76].VisStatus
    Rectangle (124,117 40x20), "P077", colour variable: DataPsgForVis[77].VisStatus
    Rectangle (164,117 40x20), "P078", colour variable: DataPsgForVis[78].VisStatus
    Rectangle (208,117 40x19), "P079", colour variable: DataPsgForVis[79].VisStatus
    Rectangle (248,117 40x20), "P080", colour variable: DataPsgForVis[80].VisStatus
    Rectangle (292,117 40x20), "P081", colour variable: DataPsgForVis[81].VisStatus
    Rectangle (332,117 40x20), "P082", colour variable: DataPsgForVis[82].VisStatus
    Rectangle (376,117 40x20), "P083", colour variable: DataPsgForVis[83].VisStatus
    Rectangle (416,117 40x20), "P084", colour variable: DataPsgForVis[85].VisStatus
    Rectangle (460,117 40x20), "P085", colour variable: DataPsgForVis[85].VisStatus
    Rectangle (500,117 40x20), "P086", colour variable: DataPsgForVis[86].VisStatus
    Rectangle (544,117 40x20), "P087", colour variable: DataPsgForVis[87].VisStatus
    Rectangle (584,117 40x20), "P088", colour variable: DataPsgForVis[88].VisStatus
    Rectangle (628,117 40x20), "P121", colour variable: DataPsgForVis[121].VisStatus
    Rectangle (668,117 40x20), "P122", colour variable: DataPsgForVis[122].VisStatus
    Rectangle (712,117 40x20), "P123", colour variable: DataPsgForVis[123].VisStatus
    Rectangle (752,117 40x20), "P124", colour variable: DataPsgForVis[124].VisStatus
    Rectangle (124,160 40x20), "P125", colour variable: DataPsgForVis[125].VisStatus
    Rectangle (164,160 40x20), "P126", colour variable: DataPsgForVis[126].VisStatus
    Rectangle (208,160 40x20), "P127", colour variable: DataPsgForVis[127].VisStatus
    Rectangle (248,160 40x20), "P128", colour variable: DataPsgForVis[128].VisStatus
    Rectangle (292,160 40x20), "P129", colour variable: DataPsgForVis[129].VisStatus
    Rectangle (332,160 40x20), "P130", colour variable: DataPsgForVis[130].VisStatus
    Rectangle (376,160 40x20), "P131", colour variable: DataPsgForVis[131].VisStatus
    Rectangle (416,160 40x20), "P132", colour variable: DataPsgForVis[132].VisStatus
    Rectangle (460,160 40x20), "P133", colour variable: DataPsgForVis[133].VisStatus
    Rectangle (500,160 40x20), "P134", colour variable: DataPsgForVis[134].VisStatus
    Rectangle (544,160 40x20), "P135", colour variable: DataPsgForVis[135].VisStatus
    Rectangle (584,160 40x20), "P136", colour variable: DataPsgForVis[136].VisStatus
    Rectangle (628,160 40x20), "P137", colour variable: DataPsgForVis[137].VisStatus
    Rectangle (668,160 40x20), "P138", colour variable: DataPsgForVis[138].VisStatus
    Rectangle (712,160 40x20), "P139", colour variable: DataPsgForVis[139].VisStatus
    Rectangle (752,160 40x20), "P140", colour variable: DataPsgForVis[140].VisStatus
    Rectangle (124,203 40x20), "P141", colour variable: DataPsgForVis[141].VisStatus
    Rectangle (164,203 40x20), "P142", colour variable: DataPsgForVis[142].VisStatus
    Rectangle (208,203 40x20), "P143", colour variable: DataPsgForVis[143].VisStatus
    Rectangle (248,203 40x20), "P144", colour variable: DataPsgForVis[144].VisStatus
    Rectangle (292,203 40x20), "P145", colour variable: DataPsgForVis[145].VisStatus
    Rectangle (332,203 40x20), "P146", colour variable: DataPsgForVis[146].VisStatus
    Rectangle (376,203 40x20), "P147", colour variable: DataPsgForVis[147].VisStatus
    Rectangle (416,203 40x20), "P148", colour variable: DataPsgForVis[148].VisStatus
    Rectangle (376,422 80x18), "ADD 28A", colour toggle: ASI02.Asi_DeviceA[28]
    Rectangle (109,524 451x21), "Timer lux"
    Rectangle (240,670 50x20), "Lux70", colour variable: DataLuxForVis[70].VisStatus
    Rectangle (290,670 40x20), "%d", text variable: DataLuxForVis[70].VisTimer, colour toggle: CronEd.CN_Sel<>CronEd.CN_Act
    Rectangle (240,710 50x20), "Lux72", colour variable: DataLuxForVis[72].VisStatus
    Rectangle (290,710 40x20), "%d", text variable: DataLuxForVis[72].VisTimer, colour toggle: CronEd.CN_Sel<>CronEd.CN_Act
    Rectangle (240,690 50x20), "Lux71", colour variable: DataLuxForVis[71].VisStatus
    Rectangle (290,690 40x20), "%d", text variable: DataLuxForVis[71].VisTimer, colour toggle: CronEd.CN_Sel<>CronEd.CN_Act
    Rectangle (221,650 19x80), "13 B", colour toggle: ASI02.Asi_DeviceB[13]
    Rectangle (240,650 50x20), "Lux69", colour variable: DataLuxForVis[69].VisStatus
    Rectangle (290,650 40x20), "%d", text variable: DataLuxForVis[69].VisTimer, colour toggle: CronEd.CN_Sel<>CronEd.CN_Act
    Rectangle (240,734 50x20), "Lux73", colour variable: DataLuxForVis[73].VisStatus
    Rectangle (290,734 40x20), "%d", text variable: DataLuxForVis[73].VisTimer, colour toggle: CronEd.CN_Sel<>CronEd.CN_Act
    Rectangle (240,754 50x20), "Lux74", colour variable: DataLuxForVis[74].VisStatus
    Rectangle (290,754 40x20), "%d", text variable: DataLuxForVis[74].VisTimer, colour toggle: CronEd.CN_Sel<>CronEd.CN_Act
    Rectangle (240,774 50x20), "Lux75", colour variable: DataLuxForVis[75].VisStatus
    Rectangle (290,774 40x20), "%d", text variable: DataLuxForVis[75].VisTimer, colour toggle: CronEd.CN_Sel<>CronEd.CN_Act
    Rectangle (240,794 50x20), "Lux76", colour variable: DataLuxForVis[76].VisStatus
    Rectangle (290,794 40x20), "%d", text variable: DataLuxForVis[76].VisTimer, colour toggle: CronEd.CN_Sel<>CronEd.CN_Act
    Rectangle (240,818 50x20), "Lux77", colour variable: DataLuxForVis[77].VisStatus
    Rectangle (290,818 40x20), "%d", text variable: DataLuxForVis[77].VisTimer, colour toggle: CronEd.CN_Sel<>CronEd.CN_Act
    Rectangle (221,734 19x80), "14 B", colour toggle: ASI02.Asi_DeviceB[14]
    Rectangle (240,838 50x20), "Lux78", colour variable: DataLuxForVis[78].VisStatus
    Rectangle (290,838 40x20), "%d", text variable: DataLuxForVis[78].VisTimer, colour toggle: CronEd.CN_Sel<>CronEd.CN_Act
    Rectangle (240,858 50x20), "Lux79", colour variable: DataLuxForVis[79].VisStatus
    Rectangle (290,858 40x20), "%d", text variable: DataLuxForVis[79].VisTimer, colour toggle: CronEd.CN_Sel<>CronEd.CN_Act
    Rectangle (240,878 50x20), "Lux80", colour variable: DataLuxForVis[80].VisStatus
    Rectangle (290,878 40x20), "%d", text variable: DataLuxForVis[80].VisTimer, colour toggle: CronEd.CN_Sel<>CronEd.CN_Act
    Rectangle (221,818 19x80), "15 B", colour toggle: ASI02.Asi_DeviceB[15]
    Rectangle (353,566 50x20), "Lux81", colour variable: DataLuxForVis[81].VisStatus
    Rectangle (403,566 40x20), "%d", text variable: DataLuxForVis[81].VisTimer, colour toggle: CronEd.CN_Sel<>CronEd.CN_Act
    Rectangle (353,586 50x20), "Lux82", colour variable: DataLuxForVis[82].VisStatus
    Rectangle (403,586 40x20), "%d", text variable: DataLuxForVis[82].VisTimer, colour toggle: CronEd.CN_Sel<>CronEd.CN_Act
    Rectangle (353,606 50x20), "Lux83", colour variable: DataLuxForVis[83].VisStatus
    Rectangle (403,606 40x20), "%d", text variable: DataLuxForVis[83].VisTimer, colour toggle: CronEd.CN_Sel<>CronEd.CN_Act
    Rectangle (353,626 50x20), "Lux84", colour variable: DataLuxForVis[84].VisStatus
    Rectangle (403,626 40x20), "%d", text variable: DataLuxForVis[84].VisTimer, colour toggle: CronEd.CN_Sel<>CronEd.CN_Act
    Rectangle (334,566 19x80), "16 B", colour toggle: ASI02.Asi_DeviceB[16]
    Rectangle (353,650 50x20), "Lux85", colour variable: DataLuxForVis[85].VisStatus
    Rectangle (403,650 40x20), "%d", text variable: DataLuxForVis[85].VisTimer, colour toggle: CronEd.CN_Sel<>CronEd.CN_Act
    Rectangle (353,670 50x20), "Lux86", colour variable: DataLuxForVis[86].VisStatus
    Rectangle (403,670 40x20), "%d", text variable: DataLuxForVis[86].VisTimer, colour toggle: CronEd.CN_Sel<>CronEd.CN_Act
    Rectangle (353,690 50x20), "Lux87", colour variable: DataLuxForVis[87].VisStatus
    Rectangle (403,690 40x20), "%d", text variable: DataLuxForVis[87].VisTimer, colour toggle: CronEd.CN_Sel<>CronEd.CN_Act
    Rectangle (353,710 50x20), "Lux88", colour variable: DataLuxForVis[88].VisStatus
    Rectangle (403,710 40x20), "%d", text variable: DataLuxForVis[88].VisTimer, colour toggle: CronEd.CN_Sel<>CronEd.CN_Act
    Rectangle (334,650 19x80), "17 B", colour toggle: ASI02.Asi_DeviceB[17]
    Rectangle (467,650 50x20), "Lux101", colour variable: DataLuxForVis[101].VisStatus
    Rectangle (517,650 40x20), "%d", text variable: DataLuxForVis[101].VisTimer, colour toggle: CronEd.CN_Sel<>CronEd.CN_Act
    Rectangle (467,670 50x20), "Lux102", colour variable: DataLuxForVis[102].VisStatus
    Rectangle (517,670 40x20), "%d", text variable: DataLuxForVis[102].VisTimer, colour toggle: CronEd.CN_Sel<>CronEd.CN_Act
    Rectangle (467,690 50x20), "Lux103", colour variable: DataLuxForVis[103].VisStatus
    Rectangle (517,690 40x20), "%d", text variable: DataLuxForVis[103].VisTimer, colour toggle: CronEd.CN_Sel<>CronEd.CN_Act
    Rectangle (467,710 50x20), "Lux104", colour variable: DataLuxForVis[104].VisStatus
    Rectangle (517,710 40x20), "%d", text variable: DataLuxForVis[104].VisTimer, colour toggle: CronEd.CN_Sel<>CronEd.CN_Act
    Rectangle (448,650 19x80), "21 B", colour toggle: ASI02.Asi_DeviceB[21]
    Rectangle (353,734 50x20), "Lux89", colour variable: DataLuxForVis[89].VisStatus
    Rectangle (403,734 40x20), "%d", text variable: DataLuxForVis[89].VisTimer, colour toggle: CronEd.CN_Sel<>CronEd.CN_Act
    Rectangle (353,754 50x20), "Lux90", colour variable: DataLuxForVis[90].VisStatus
    Rectangle (403,754 40x20), "%d", text variable: DataLuxForVis[90].VisTimer, colour toggle: CronEd.CN_Sel<>CronEd.CN_Act
    Rectangle (353,774 50x20), "Lux91", colour variable: DataLuxForVis[91].VisStatus
    Rectangle (403,774 40x20), "%d", text variable: DataLuxForVis[91].VisTimer, colour toggle: CronEd.CN_Sel<>CronEd.CN_Act
    Rectangle (353,794 50x20), "Lux92", colour variable: DataLuxForVis[92].VisStatus
    Rectangle (403,794 40x20), "%d", text variable: DataLuxForVis[92].VisTimer, colour toggle: CronEd.CN_Sel<>CronEd.CN_Act
    Rectangle (334,734 19x80), "18 B", colour toggle: ASI02.Asi_DeviceB[18]
    Rectangle (353,818 50x20), "Lux93", colour variable: DataLuxForVis[93].VisStatus
    Rectangle (403,818 40x20), "%d", text variable: DataLuxForVis[93].VisTimer, colour toggle: CronEd.CN_Sel<>CronEd.CN_Act
    Rectangle (353,838 50x20), "Lux94", colour variable: DataLuxForVis[94].VisStatus
    Rectangle (403,838 40x20), "%d", text variable: DataLuxForVis[94].VisTimer, colour toggle: CronEd.CN_Sel<>CronEd.CN_Act
    Rectangle (353,858 50x20), "Lux95", colour variable: DataLuxForVis[95].VisStatus
    Rectangle (403,858 40x20), "%d", text variable: DataLuxForVis[95].VisTimer, colour toggle: CronEd.CN_Sel<>CronEd.CN_Act
    Rectangle (353,878 50x20), "Lux96", colour variable: DataLuxForVis[96].VisStatus
    Rectangle (403,878 40x20), "%d", text variable: DataLuxForVis[96].VisTimer, colour toggle: CronEd.CN_Sel<>CronEd.CN_Act
    Rectangle (334,818 19x80), "19 B", colour toggle: ASI02.Asi_DeviceB[19]
    Rectangle (467,566 50x20), "Lux97", colour variable: DataLuxForVis[97].VisStatus
    Rectangle (517,566 40x20), "%d", text variable: DataLuxForVis[97].VisTimer, colour toggle: CronEd.CN_Sel<>CronEd.CN_Act
    Rectangle (467,586 50x20), "Lux98", colour variable: DataLuxForVis[98].VisStatus
    Rectangle (517,586 40x20), "%d", text variable: DataLuxForVis[98].VisTimer, colour toggle: CronEd.CN_Sel<>CronEd.CN_Act
    Rectangle (467,606 50x20), "Lux99", colour variable: DataLuxForVis[99].VisStatus
    Rectangle (517,606 40x20), "%d", text variable: DataLuxForVis[99].VisTimer, colour toggle: CronEd.CN_Sel<>CronEd.CN_Act
    Rectangle (467,626 50x20), "Lux100", colour variable: DataLuxForVis[100].VisStatus
    Rectangle (517,626 40x20), "%d", text variable: DataLuxForVis[100].VisTimer, colour toggle: CronEd.CN_Sel<>CronEd.CN_Act
    Rectangle (448,566 19x80), "20 B", colour toggle: ASI02.Asi_DeviceB[20]
    Rectangle (128,566 50x20), "Lux49", colour variable: DataLuxForVis[49].VisStatus
    Rectangle (178,566 40x20), "%d", text variable: DataLuxForVis[49].VisTimer, colour toggle: CronEd.CN_Sel<>CronEd.CN_Act
    Rectangle (128,586 50x20), "Lux50", colour variable: DataLuxForVis[50].VisStatus
    Rectangle (178,586 40x20), "%d", text variable: DataLuxForVis[50].VisTimer, colour toggle: CronEd.CN_Sel<>CronEd.CN_Act
    Rectangle (128,606 50x20), "Lux51", colour variable: DataLuxForVis[51].VisStatus
    Rectangle (178,606 40x20), "%d", text variable: DataLuxForVis[51].VisTimer, colour toggle: CronEd.CN_Sel<>CronEd.CN_Act
    Rectangle (128,626 50x20), "Lux52", colour variable: DataLuxForVis[52].VisStatus
    Rectangle (178,626 40x20), "%d", text variable: DataLuxForVis[52].VisTimer, colour toggle: CronEd.CN_Sel<>CronEd.CN_Act
    Rectangle (109,566 19x80), "08 B", colour toggle: ASI02.Asi_DeviceB[8]
    Rectangle (128,650 50x20), "Lux53", colour variable: DataLuxForVis[53].VisStatus
    Rectangle (178,650 40x20), "%d", text variable: DataLuxForVis[53].VisTimer, colour toggle: CronEd.CN_Sel<>CronEd.CN_Act
    Rectangle (128,670 50x20), "Lux54", colour variable: DataLuxForVis[54].VisStatus
    Rectangle (178,670 40x20), "%d", text variable: DataLuxForVis[54].VisTimer, colour toggle: CronEd.CN_Sel<>CronEd.CN_Act
    Rectangle (128,690 50x20), "Lux55", colour variable: DataLuxForVis[55].VisStatus
    Rectangle (178,690 40x20), "%d", text variable: DataLuxForVis[55].VisTimer, colour toggle: CronEd.CN_Sel<>CronEd.CN_Act
    Rectangle (128,710 50x20), "Lux56", colour variable: DataLuxForVis[56].VisStatus
    Rectangle (178,710 40x20), "%d", text variable: DataLuxForVis[56].VisTimer, colour toggle: CronEd.CN_Sel<>CronEd.CN_Act
    Rectangle (109,650 19x80), "09 B", colour toggle: ASI02.Asi_DeviceB[9]
    Rectangle (128,734 50x20), "Lux57", colour variable: DataLuxForVis[57].VisStatus
    Rectangle (178,734 40x20), "%d", text variable: DataLuxForVis[57].VisTimer, colour toggle: CronEd.CN_Sel<>CronEd.CN_Act
    Rectangle (128,754 50x20), "Lux58", colour variable: DataLuxForVis[58].VisStatus
    Rectangle (178,754 40x20), "%d", text variable: DataLuxForVis[58].VisTimer, colour toggle: CronEd.CN_Sel<>CronEd.CN_Act
    Rectangle (128,774 50x20), "Lux59", colour variable: DataLuxForVis[59].VisStatus
    Rectangle (178,774 40x20), "%d", text variable: DataLuxForVis[59].VisTimer, colour toggle: CronEd.CN_Sel<>CronEd.CN_Act
    Rectangle (128,794 50x20), "Lux60", colour variable: DataLuxForVis[60].VisStatus
    Rectangle (178,794 40x20), "%d", text variable: DataLuxForVis[60].VisTimer, colour toggle: CronEd.CN_Sel<>CronEd.CN_Act
        OnMouseDown: write the text variable via Edit, min 10, max 32760, title '1'
    Rectangle (109,734 19x80), "10 B", colour toggle: ASI02.Asi_DeviceB[10]
    Rectangle (128,818 50x20), "Lux61", colour variable: DataLuxForVis[61].VisStatus
    Rectangle (178,818 40x20), "%d", text variable: DataLuxForVis[61].VisTimer, colour toggle: CronEd.CN_Sel<>CronEd.CN_Act
    Rectangle (128,838 50x20), "Lux62", colour variable: DataLuxForVis[62].VisStatus
    Rectangle (178,838 40x20), "%d", text variable: DataLuxForVis[62].VisTimer, colour toggle: CronEd.CN_Sel<>CronEd.CN_Act
    Rectangle (128,858 50x20), "Lux63", colour variable: DataLuxForVis[63].VisStatus
    Rectangle (178,858 40x20), "%d", text variable: DataLuxForVis[63].VisTimer, colour toggle: CronEd.CN_Sel<>CronEd.CN_Act
    Rectangle (128,878 50x20), "Lux64", colour variable: DataLuxForVis[64].VisStatus
    Rectangle (178,878 40x20), "%d", text variable: DataLuxForVis[64].VisTimer, colour toggle: CronEd.CN_Sel<>CronEd.CN_Act
    Rectangle (109,818 19x80), "11 B", colour toggle: ASI02.Asi_DeviceB[11]
    Rectangle (240,566 50x20), "Lux65", colour variable: DataLuxForVis[65].VisStatus
    Rectangle (290,566 40x20), "%d", text variable: DataLuxForVis[65].VisTimer, colour toggle: CronEd.CN_Sel<>CronEd.CN_Act
    Rectangle (240,586 50x20), "Lux66", colour variable: DataLuxForVis[66].VisStatus
    Rectangle (290,586 40x20), "%d", text variable: DataLuxForVis[66].VisTimer, colour toggle: CronEd.CN_Sel<>CronEd.CN_Act
    Rectangle (240,606 50x20), "Lux67", colour variable: DataLuxForVis[67].VisStatus
    Rectangle (290,606 40x20), "%d", text variable: DataLuxForVis[67].VisTimer, colour toggle: CronEd.CN_Sel<>CronEd.CN_Act
    Rectangle (240,626 50x20), "Lux68", colour variable: DataLuxForVis[68].VisStatus
    Rectangle (290,626 40x20), "%d", text variable: DataLuxForVis[68].VisTimer, colour toggle: CronEd.CN_Sel<>CronEd.CN_Act
    Rectangle (221,566 19x80), "12 B", colour toggle: ASI02.Asi_DeviceB[12]
    Rectangle (109,547 451x17), "ASI 2"
    Rectangle (108,936 115x17), "ASI 1"
    Rectangle (108,912 467x21), "Crono lux"
    Rectangle (133,955 50x20), "Lux043", colour variable: DataLuxForVis[43].VisStatus
    Rectangle (183,955 40x20), "%d", text variable: DataLuxForVis[43].VisMod, colour toggle: CronEd.CN_Sel<>CronEd.CN_Act
    Rectangle (133,975 50x20), "Lux044", colour variable: DataLuxForVis[44].VisStatus
    Rectangle (183,975 40x20), "%d", text variable: DataLuxForVis[44].VisMod, colour toggle: CronEd.CN_Sel<>CronEd.CN_Act
    Rectangle (133,995 50x20), "Lux045", colour variable: DataLuxForVis[45].VisStatus
    Rectangle (183,995 40x20), "%d", text variable: DataLuxForVis[45].VisMod, colour toggle: CronEd.CN_Sel<>CronEd.CN_Act
    Rectangle (108,955 25x20), "29A", colour toggle: ASI01.Asi_DeviceB[29]
    Rectangle (108,975 25x20), "30A", colour toggle: ASI01.Asi_DeviceB[30]
    Rectangle (108,995 25x20), "31A", colour toggle: ASI01.Asi_DeviceB[31]
    Rectangle (226,936 349x17), "ASI 2"
    Rectangle (251,995 50x20), "Lux15", colour variable: DataLuxForVis[15].VisStatus
    Rectangle (301,995 40x20), "%d", text variable: DataLuxForVis[15].VisMod, colour toggle: CronEd.CN_Sel<>CronEd.CN_Act
    Rectangle (226,995 25x20), "02B", colour toggle: ASI02.Asi_DeviceB[2]
    Rectangle (226,1015 25x20), "02B", colour toggle: ASI02.Asi_DeviceB[2]
    Rectangle (251,1015 50x20), "Lux16", colour variable: DataLuxForVis[16].VisStatus
    Rectangle (301,1015 40x20), "%d", text variable: DataLuxForVis[16].VisMod, colour toggle: CronEd.CN_Sel<>CronEd.CN_Act
    Rectangle (226,1035 25x20), "03B", colour toggle: ASI02.Asi_DeviceB[3]
    Rectangle (251,1035 50x20), "Lux17", colour variable: DataLuxForVis[17].VisStatus
    Rectangle (301,1035 40x20), "%d", text variable: DataLuxForVis[17].VisMod, colour toggle: CronEd.CN_Sel<>CronEd.CN_Act
    Rectangle (226,1055 25x20), "03B", colour toggle: ASI02.Asi_DeviceB[3]
    Rectangle (251,1055 50x20), "Lux18", colour variable: DataLuxForVis[18].VisStatus
    Rectangle (301,1055 40x20), "%d", text variable: DataLuxForVis[18].VisMod, colour toggle: CronEd.CN_Sel<>CronEd.CN_Act
    Rectangle (251,1075 50x20), "Lux19", colour variable: DataLuxForVis[19].VisStatus
    Rectangle (301,1075 40x20), "%d", text variable: DataLuxForVis[19].VisMod, colour toggle: CronEd.CN_Sel<>CronEd.CN_Act
    Rectangle (226,1075 25x20), "04B", colour toggle: ASI02.Asi_DeviceB[4]
    Rectangle (226,1095 25x20), "04B", colour toggle: ASI02.Asi_DeviceB[4]
    Rectangle (251,1095 50x20), "Lux20", colour variable: DataLuxForVis[20].VisStatus
    Rectangle (301,1095 40x20), "%d", text variable: DataLuxForVis[20].VisMod, colour toggle: CronEd.CN_Sel<>CronEd.CN_Act
    Rectangle (226,1115 25x20), "05B", colour toggle: ASI02.Asi_DeviceB[5]
    Rectangle (251,1115 50x20), "Lux21", colour variable: DataLuxForVis[21].VisStatus
    Rectangle (301,1115 40x20), "%d", text variable: DataLuxForVis[21].VisMod, colour toggle: CronEd.CN_Sel<>CronEd.CN_Act
    Rectangle (226,1135 25x20), "05B", colour toggle: ASI02.Asi_DeviceB[5]
    Rectangle (251,1135 50x20), "Lux22", colour variable: DataLuxForVis[22].VisStatus
    Rectangle (301,1135 40x20), "%d", text variable: DataLuxForVis[22].VisMod, colour toggle: CronEd.CN_Sel<>CronEd.CN_Act
    Rectangle (251,1155 50x20), "Lux23", colour variable: DataLuxForVis[23].VisStatus
    Rectangle (301,1155 40x20), "%d", text variable: DataLuxForVis[23].VisMod, colour toggle: CronEd.CN_Sel<>CronEd.CN_Act
    Rectangle (226,1155 25x20), "06B", colour toggle: ASI02.Asi_DeviceB[6]
    Rectangle (226,1175 25x20), "06B", colour toggle: ASI02.Asi_DeviceB[6]
    Rectangle (251,1175 50x20), "Lux24", colour variable: DataLuxForVis[24].VisStatus
    Rectangle (301,1175 40x20), "%d", text variable: DataLuxForVis[24].VisMod, colour toggle: CronEd.CN_Sel<>CronEd.CN_Act
    Rectangle (344,955 25x20), "29A", colour toggle: ASI02.Asi_DeviceA[29]
    Rectangle (369,955 50x20), "Lux01", colour variable: DataLuxForVis[1].VisStatus
    Rectangle (419,955 40x20), "%d", text variable: DataLuxForVis[1].VisMod, colour toggle: CronEd.CN_Sel<>CronEd.CN_Act
    Rectangle (344,975 25x20), "29A", colour toggle: ASI02.Asi_DeviceA[29]
    Rectangle (369,975 50x20), "Lux02", colour variable: DataLuxForVis[2].VisStatus
    Rectangle (419,975 40x20), "%d", text variable: DataLuxForVis[2].VisMod, colour toggle: CronEd.CN_Sel<>CronEd.CN_Act
    Rectangle (369,995 50x20), "Lux03", colour variable: DataLuxForVis[3].VisStatus
    Rectangle (419,995 40x20), "%d", text variable: DataLuxForVis[3].VisMod, colour toggle: CronEd.CN_Sel<>CronEd.CN_Act
    Rectangle (344,995 25x20), "30A", colour toggle: ASI02.Asi_DeviceA[30]
    Rectangle (344,1015 25x20), "30A", colour toggle: ASI02.Asi_DeviceA[30]
    Rectangle (369,1015 50x20), "Lux04", colour variable: DataLuxForVis[04].VisStatus
    Rectangle (419,1015 40x20), "%d", text variable: DataLuxForVis[4].VisMod, colour toggle: CronEd.CN_Sel<>CronEd.CN_Act
    Rectangle (344,1035 25x20), "31A", colour toggle: ASI02.Asi_DeviceA[31]
    Rectangle (369,1035 50x20), "Lux05", colour variable: DataLuxForVis[05].VisStatus
    Rectangle (419,1035 40x20), "%d", text variable: DataLuxForVis[5].VisMod, colour toggle: CronEd.CN_Sel<>CronEd.CN_Act
    Rectangle (344,1055 25x20), "31A", colour toggle: ASI02.Asi_DeviceA[31]
    Rectangle (369,1055 50x20), "Lux06", colour variable: DataLuxForVis[06].VisStatus
    Rectangle (419,1055 40x20), "%d", text variable: DataLuxForVis[6].VisMod, colour toggle: CronEd.CN_Sel<>CronEd.CN_Act
    Rectangle (124,56 80x18), "ADD 01A", colour toggle: ASI01.Asi_DeviceA[1]
    Rectangle (208,56 80x18), "ADD 02A", colour toggle: ASI01.Asi_DeviceA[2]
    Rectangle (292,56 80x18), "ADD 03A", colour toggle: ASI01.Asi_DeviceA[3]
    Rectangle (376,56 80x18), "ADD 04A", colour toggle: ASI01.Asi_DeviceA[4]
    Rectangle (460,56 80x18), "ADD 05A", colour toggle: ASI01.Asi_DeviceA[5]
    Rectangle (544,56 80x18), "ADD 06A", colour toggle: ASI01.Asi_DeviceA[6]
    Rectangle (628,56 80x18), "ADD 07A", colour toggle: ASI01.Asi_DeviceA[7]
    Rectangle (712,56 80x18), "ADD 08A", colour toggle: ASI01.Asi_DeviceA[8]
    Rectangle (712,99 80x18), "ADD 16A", colour toggle: ASI01.Asi_DeviceA[16]
    Rectangle (124,99 80x18), "ADD 09A", colour toggle: ASI01.Asi_DeviceA[9]
    Rectangle (208,99 80x18), "ADD 10A", colour toggle: ASI01.Asi_DeviceA[10]
    Rectangle (292,99 80x18), "ADD 11A", colour toggle: ASI01.Asi_DeviceA[11]
    Rectangle (376,99 80x18), "ADD 12A", colour toggle: ASI01.Asi_DeviceA[12]
    Rectangle (460,99 80x18), "ADD 13A", colour toggle: ASI01.Asi_DeviceA[13]
    Rectangle (544,99 80x18), "ADD 14A", colour toggle: ASI01.Asi_DeviceA[14]
    Rectangle (628,99 80x18), "ADD 15A", colour toggle: ASI01.Asi_DeviceA[15]
    Rectangle (712,142 80x18), "ADD 24A", colour toggle: ASI01.Asi_DeviceA[24]
    Rectangle (124,142 80x18), "ADD 17A", colour toggle: ASI01.Asi_DeviceA[17]
    Rectangle (208,142 80x18), "ADD 18A", colour toggle: ASI01.Asi_DeviceA[18]
    Rectangle (292,142 80x18), "ADD 19A", colour toggle: ASI01.Asi_DeviceA[19]
    Rectangle (376,142 80x18), "ADD 20A", colour toggle: ASI01.Asi_DeviceA[20]
    Rectangle (460,142 80x18), "ADD 21A", colour toggle: ASI01.Asi_DeviceA[21]
    Rectangle (544,142 80x18), "ADD 22A", colour toggle: ASI01.Asi_DeviceA[22]
    Rectangle (628,142 80x18), "ADD 23A", colour toggle: ASI01.Asi_DeviceA[23]
    Rectangle (124,185 80x18), "ADD 25A", colour toggle: ASI01.Asi_DeviceA[25]
    Rectangle (208,185 80x18), "ADD 26A", colour toggle: ASI01.Asi_DeviceA[26]
    Rectangle (292,185 80x18), "ADD 27A", colour toggle: ASI01.Asi_DeviceA[27]
    Rectangle (124,311 40x20), "P001", invisible if: FALSE, colour variable: DataPsgForVis[1].VisStatus
    Rectangle (164,311 40x20), "P002", colour variable: DataPsgForVis[02].VisStatus
    Rectangle (208,311 40x20), "P003", colour variable: DataPsgForVis[03].VisStatus
    Rectangle (248,311 40x20), "P004", colour variable: DataPsgForVis[04].VisStatus
    Rectangle (292,311 40x20), "P005", colour variable: DataPsgForVis[05].VisStatus
    Rectangle (332,311 40x20), "P006", colour variable: DataPsgForVis[06].VisStatus
    Rectangle (376,311 40x20), "P007", colour variable: DataPsgForVis[07].VisStatus
    Rectangle (416,311 40x20), "P008", colour variable: DataPsgForVis[08].VisStatus
    Rectangle (460,311 40x20), "P009", colour variable: DataPsgForVis[09].VisStatus
    Rectangle (500,311 40x20), "P010", colour variable: DataPsgForVis[10].VisStatus
    Rectangle (544,311 40x20), "P011", colour variable: DataPsgForVis[11].VisStatus
    Rectangle (584,311 40x20), "P012", colour variable: DataPsgForVis[12].VisStatus
    Rectangle (628,311 40x20), "P013", colour variable: DataPsgForVis[13].VisStatus
    Rectangle (668,311 40x20), "P014", colour variable: DataPsgForVis[14].VisStatus
    Rectangle (712,311 40x20), "P015", colour variable: DataPsgForVis[15].VisStatus
    Rectangle (752,311 40x20), "P016", colour variable: DataPsgForVis[16].VisStatus
    Rectangle (712,354 40x20), "P183", colour variable: DataPsgForVis[183].VisStatus
    Rectangle (752,354 40x20), "P184", colour variable: DataPsgForVis[184].VisStatus
    Rectangle (124,354 40x20), "P017", colour variable: DataPsgForVis[17].VisStatus
    Rectangle (164,354 40x20), "P018", colour variable: DataPsgForVis[18].VisStatus
    Rectangle (208,354 40x20), "P019", colour variable: DataPsgForVis[19].VisStatus
    Rectangle (248,354 40x20), "P020", colour variable: DataPsgForVis[20].VisStatus
    Rectangle (292,354 40x20), "P021", colour variable: DataPsgForVis[21].VisStatus
    Rectangle (332,354 40x20), "P022", colour variable: DataPsgForVis[22].VisStatus
    Rectangle (376,354 40x20), "P023", colour variable: DataPsgForVis[23].VisStatus
    Rectangle (416,354 40x20), "P024", colour variable: DataPsgForVis[24].VisStatus
    Rectangle (460,354 40x20), "P025", colour variable: DataPsgForVis[25].VisStatus
    Rectangle (500,354 40x20), "P026", colour variable: DataPsgForVis[26].VisStatus
    Rectangle (544,354 40x20), "P027", colour variable: DataPsgForVis[27].VisStatus
    Rectangle (584,354 40x20), "P028", colour variable: DataPsgForVis[28].VisStatus
    Rectangle (628,354 40x20), "P181", colour variable: DataPsgForVis[181].VisStatus
    Rectangle (668,354 40x20), "P182", colour variable: DataPsgForVis[182].VisStatus
    Rectangle (712,397 40x20), "P199", colour variable: DataPsgForVis[199].VisStatus
    Rectangle (752,397 40x20), "P200", colour variable: DataPsgForVis[200].VisStatus
    Rectangle (124,397 40x20), "P185", colour variable: DataPsgForVis[185].VisStatus
    Rectangle (164,397 40x20), "P186", colour variable: DataPsgForVis[186].VisStatus
    Rectangle (208,397 40x20), "P187", colour variable: DataPsgForVis[187].VisStatus
    Rectangle (248,397 40x20), "P188", colour variable: DataPsgForVis[188].VisStatus
    Rectangle (292,397 40x20), "P189", colour variable: DataPsgForVis[189].VisStatus
    Rectangle (332,397 40x20), "P190", colour variable: DataPsgForVis[190].VisStatus
    Rectangle (376,397 40x20), "P191", colour variable: DataPsgForVis[191].VisStatus
    Rectangle (416,397 40x20), "P192", colour variable: DataPsgForVis[192].VisStatus
    Rectangle (460,397 40x20), "P193", colour variable: DataPsgForVis[193].VisStatus
    Rectangle (500,397 40x20), "P194", colour variable: DataPsgForVis[194].VisStatus
    Rectangle (544,397 40x20), "P195", colour variable: DataPsgForVis[195].VisStatus
    Rectangle (584,397 40x20), "P196", colour variable: DataPsgForVis[196].VisStatus
    Rectangle (628,397 40x20), "P197", colour variable: DataPsgForVis[197].VisStatus
    Rectangle (668,397 40x20), "P198", colour variable: DataPsgForVis[198].VisStatus
    Rectangle (124,440 40x20), "P201", colour variable: DataPsgForVis[201].VisStatus
    Rectangle (164,440 40x20), "P202", colour variable: DataPsgForVis[202].VisStatus
    Rectangle (208,440 40x20), "P203", colour variable: DataPsgForVis[203].VisStatus
    Rectangle (248,440 40x20), "P204", colour variable: DataPsgForVis[204].VisStatus
    Rectangle (292,440 40x20), "P205", colour variable: DataPsgForVis[205].VisStatus
    Rectangle (332,440 40x20), "P206", colour variable: DataPsgForVis[206].VisStatus
    Rectangle (376,440 40x20), "P207", colour variable: DataPsgForVis[207].VisStatus
    Rectangle (416,440 40x20), "P208", colour variable: DataPsgForVis[208].VisStatus
    Rectangle (376,185 80x18), "ADD 28A", colour toggle: ASI01.Asi_DeviceA[28]
    Rectangle (568,524 156x21), "Timer lux modify"
    Rectangle (568,547 156x112)
    Rectangle (574,553 60x20), "LUX Nr."
    Rectangle (634,553 40x20), "%d", text variable: PLC_PRG.TimerLuxSelected
        OnMouseDown: write the text variable via Edit, min 1, max LUXM_MAX_ID, title '1'
    Rectangle (634,574 40x20), "%d", text variable: DataLuxForVis[PLC_PRG.TimerLuxSelected].VisTimer
    Rectangle (574,574 60x20), "Timer (s)"
    Button (574,632 137x20), "Change timer"
        OnMouseClick:  ToggleVariable=PLC_PRG.VisModify_T_Lux
    Rectangle (672,603 40x20), "%d", text variable: PLC_PRG.TimerLuxValue
        OnMouseDown: write the text variable via Edit, min 1, max 65000, title '1'
    Rectangle (574,603 97x20), "New value (s)"
    Rectangle (584,913 152x21), "On/Off Lux"
    Group (584,937 152x112)
        Rectangle (0,0 152x112)
        Rectangle (3,4 60x20), "LUX Nr."
        Rectangle (63,4 40x20), "%d", text variable: PLC_PRG.VisLuxOnOffSelected
            OnMouseDown: write the text variable via Edit, min 1, max LUXM_MAX_ID, title '1'
        Button (8,86 137x20), "Change mode"
            OnMouseClick:  ToggleVariable=PLC_PRG.VisModify_Man_Lux
        Rectangle (3,30 39x53), "Aut Man"
        DipSwitch (33,39 40x43), variable: PLC_PRG.VisValueManAut, behaviour: TOGGLE, style: Switch-DipSwitch-Gray
        Rectangle (75,30 39x53), "On Off"
        DipSwitch (104,39 40x43), variable: PLC_PRG.VisValueManOnOff, behaviour: TOGGLE, style: Switch-DipSwitch-Gray
    Rectangle (585,1056 107x95), "Mode: 00 - Man Off 01 - Man On 02 - Aut Cron 03 - Aut Timer"
    Button (731,11 60x30), "Crono"
        OnMouseUp:  Assign=VIS_CHONOEDITOR, Type=Assignment
    Rectangle (125,11 586x30), "%s === Visualization", text variable: Plant_NAME
    Rectangle (568,670 156x52), "Green - OK, Off Light Green - OK, On Red - Asi slave Error", invisible if: 0
    Rectangle (2,80 119x32), "Green - ASi OK Yellow - Asi Warning", invisible if: 0
    Rectangle (251,955 50x20), "Lux13", colour variable: DataLuxForVis[13].VisStatus
    Rectangle (301,955 40x20), "%d", text variable: DataLuxForVis[13].VisMod, colour toggle: CronEd.CN_Sel<>CronEd.CN_Act
    Rectangle (226,955 25x20), "01B", colour toggle: ASI02.Asi_DeviceB[1]
    Rectangle (226,975 25x20), "01B", colour toggle: ASI02.Asi_DeviceB[1]
    Rectangle (251,975 50x20), "Lux14", colour variable: DataLuxForVis[14].VisStatus
    Rectangle (301,975 40x20), "%d", text variable: DataLuxForVis[14].VisMod, colour toggle: CronEd.CN_Sel<>CronEd.CN_Act
    Rectangle (251,1195 50x20), "Lux25", colour variable: DataLuxForVis[25].VisStatus
    Rectangle (301,1195 40x20), "%d", text variable: DataLuxForVis[25].VisMod, colour toggle: CronEd.CN_Sel<>CronEd.CN_Act
    Rectangle (226,1195 25x20), "07B", colour toggle: ASI02.Asi_DeviceB[7]
    Rectangle (226,1215 25x20), "07B", colour toggle: ASI02.Asi_DeviceB[7]
    Rectangle (251,1215 50x20), "Lux26", colour variable: DataLuxForVis[26].VisStatus
    Rectangle (301,1215 40x20), "%d", text variable: DataLuxForVis[26].VisMod, colour toggle: CronEd.CN_Sel<>CronEd.CN_Act
END_VISUALIZATION
